LIN {X 0,Y 141.278,Z 230.592,A -85,B 0,C 180,E1 -25855.05,E2 -25855.05} C_VEL
LIN {X 0,Y 135.258,Z 217.256,A -85,B 0,C 180,E1 -25857.958,E2 -25857.958} C_VEL
LIN {X 0,Y 129.274,Z 206.453,A -85,B 0,C 180,E1 -25861.051,E2 -25861.051} C_VEL
LIN {X 0,Y 124.836,Z 199.374,A -85,B 0,C 180,E1 -25863.554,E2 -25863.554} C_VEL
LIN {X 0,Y 120.846,Z 193.414,A -85,B 0,C 180,E1 -25866.03,E2 -25866.03} C_VEL
LIN {X 0,Y 118.527,Z 190.076,A -85,B 0,C 180,E1 -25867.593,E2 -25867.593} C_VEL
LIN {X 0,Y 118.058,Z 189.3,A -85,B 0,C 180,E1 -25867.932,E2 -25867.932} C_VEL
LIN {X 0,Y 115.859,Z 187.104,A -85,B 0,C 180,E1 -25869.449,E2 -25869.449} C_VEL
LIN {X 0,Y 114.927,Z 184.823,A -85,B 0,C 180,E1 -25870.265,E2 -25870.265} C_VEL
LIN {X 0,Y 114.809,Z 184.184,A -85,B 0,C 180,E1 -25870.536,E2 -25870.536} C_VEL
LIN {X 0,Y 114.767,Z 184.142,A -85,B 0,C 180,E1 -25877.657,E2 -25877.657} C_VEL
LIN {X 0,Y 114.783,Z 184.185,A -85,B 0,C 180,E1 -25882.749,E2 -25882.749} C_VEL
LIN {X 0,Y 114.839,Z 184.117,A -85,B 0,C 180,E1 -25888.959,E2 -25888.959} C_VEL
LIN {X 0,Y 114.899,Z 184.166,A -85,B 0,C 180,E1 -25896.566,E2 -25896.566} C_VEL
LIN {X 0,Y 114.963,Z 184.147,A -85,B 0,C 180,E1 -25902.204,E2 -25902.204} C_VEL
LIN {X 0,Y 115.306,Z 184.11,A -85,B 0,C 180,E1 -25909.466,E2 -25909.466} C_VEL
LIN {X 0,Y 115.487,Z 184.099,A -85,B 0,C 180,E1 -25916.513,E2 -25916.513} C_VEL
LIN {X 0,Y 115.951,Z 184.025,A -85,B 0,C 180,E1 -25920.002,E2 -25920.002} C_VEL
LIN {X 0,Y 115.351,Z 184.103,A -85,B 0,C 180,E1 -25927.001,E2 -25927.001} C_VEL
LIN {X 0,Y 115.207,Z 184.136,A -85,B 0,C 180,E1 -25932.559,E2 -25932.559} C_VEL
LIN {X 0,Y 114.969,Z 184.154,A -85,B 0,C 180,E1 -25937.799,E2 -25937.799} C_VEL
LIN {X 0,Y 114.914,Z 184.172,A -85,B 0,C 180,E1 -25943.451,E2 -25943.451} C_VEL
LIN {X 0,Y 114.863,Z 184.178,A -85,B 0,C 180,E1 -25949.058,E2 -25949.058} C_VEL
LIN {X 0,Y 115.85,Z 186.976,A -85,B 0,C 180,E1 -25950.008,E2 -25950.008} C_VEL
LIN {X 0,Y 117.94,Z 189.165,A -85,B 0,C 180,E1 -25951.46,E2 -25951.46} C_VEL
LIN {X 0,Y 118.811,Z 190.602,A -85,B 0,C 180,E1 -25952.087,E2 -25952.087} C_VEL
LIN {X 0,Y 121.086,Z 193.68,A -85,B 0,C 180,E1 -25953.59,E2 -25953.59} C_VEL
LIN {X 0,Y 126.955,Z 202.682,A -85,B 0,C 180,E1 -25957.142,E2 -25957.142} C_VEL
LIN {X 0,Y 130.736,Z 209.225,A -85,B 0,C 180,E1 -25959.227,E2 -25959.227} C_VEL
LIN {X 0,Y 135.81,Z 221.695,A -85,B 0,C 180,E1 -25962.03,E2 -25962.03} C_VEL
LIN {X 0,Y 139.584,Z 233.149,A -85,B 0,C 180,E1 -25964.065,E2 -25964.065} C_VEL
LIN {X 0,Y 140.517,Z 245.678,A -85,B 0,C 180,E1 -25965.174,E2 -25965.174} C_VEL
LIN {X 0,Y 137.592,Z 288.137,A -85,B 0,C 180,E1 -25967.172,E2 -25967.172} C_VEL
LIN {X 0,Y 135.71,Z 301.694,A -85,B 0,C 180,E1 -25968.306,E2 -25968.306} C_VEL
LIN {X 0,Y 133.388,Z 313.543,A -85,B 0,C 180,E1 -25969.801,E2 -25969.801} C_VEL
LIN {X 0,Y 130.614,Z 324.787,A -85,B 0,C 180,E1 -25971.772,E2 -25971.772} C_VEL
LIN {X 0,Y 127.55,Z 335.152,A -85,B 0,C 180,E1 -25974.165,E2 -25974.165} C_VEL
LIN {X 0,Y 124.027,Z 345.896,A -85,B 0,C 180,E1 -25977.43,E2 -25977.43} C_VEL
LIN {X 0,Y 121.167,Z 354.142,A -85,B 0,C 180,E1 -25980.656,E2 -25980.656} C_VEL
LIN {X 0,Y 117.858,Z 363.477,A -85,B 0,C 180,E1 -25985.328,E2 -25985.328} C_VEL
LIN {X 0,Y 115.267,Z 371.169,A -85,B 0,C 180,E1 -25990.406,E2 -25990.406} C_VEL
LIN {X 0,Y 113.501,Z 377.329,A -85,B 0,C 180,E1 -25995.659,E2 -25995.659} C_VEL
LIN {X 0,Y 112.596,Z 382.185,A -85,B 0,C 180,E1 -26001.022,E2 -26001.022} C_VEL
LIN {X 0,Y 112.341,Z 385.87,A -85,B 0,C 180,E1 -26006.413,E2 -26006.413} C_VEL
LIN {X 0,Y 112.454,Z 387.919,A -85,B 0,C 180,E1 -26010.362,E2 -26010.362} C_VEL
LIN {X 0,Y 112.336,Z 389.142,A -85,B 0,C 180,E1 -26013.586,E2 -26013.586} C_VEL
LIN {X 0,Y 112.831,Z 390.682,A -85,B 0,C 180,E1 -26020.769,E2 -26020.769} C_VEL
LIN {X 0,Y 114.797,Z 390.713,A -85,B 0,C 180,E1 -26027.824,E2 -26027.824} C_VEL
LIN {X 0,Y 118.532,Z 389.166,A -85,B 0,C 180,E1 -26034.522,E2 -26034.522} C_VEL
LIN {X 0,Y 123.893,Z 386.089,A -85,B 0,C 180,E1 -26040.699,E2 -26040.699} C_VEL
LIN {X 0,Y 128.757,Z 382.601,A -85,B 0,C 180,E1 -26045.037,E2 -26045.037} C_VEL
LIN {X 0,Y 135.201,Z 377.315,A -85,B 0,C 180,E1 -26049.537,E2 -26049.537} C_VEL
LIN {X 0,Y 141.582,Z 371.476,A -85,B 0,C 180,E1 -26053.042,E2 -26053.042} C_VEL
LIN {X 0,Y 145.984,Z 367,A -85,B 0,C 180,E1 -26055.088,E2 -26055.088} C_VEL
LIN {X 0,Y 148.771,Z 363.579,A -85,B 0,C 180,E1 -26056.614,E2 -26056.614} C_VEL
LIN {X 0,Y 151.909,Z 357.771,A -85,B 0,C 180,E1 -26059.441,E2 -26059.441} C_VEL
LIN {X 0,Y 155.058,Z 351.474,A -85,B 0,C 180,E1 -26062.04,E2 -26062.04} C_VEL
LIN {X 0,Y 157.739,Z 347.223,A -85,B 0,C 180,E1 -26063.181,E2 -26063.181} C_VEL
LIN {X 0,Y 164.092,Z 337.097,A -85,B 0,C 180,E1 -26064.996,E2 -26064.996} C_VEL
LIN {X 0,Y 169.797,Z 326.151,A -85,B 0,C 180,E1 -26066.406,E2 -26066.406} C_VEL
LIN {X 0,Y 174.86,Z 313.961,A -85,B 0,C 180,E1 -26067.569,E2 -26067.569} C_VEL
LIN {X 0,Y 178.951,Z 301.013,A -85,B 0,C 180,E1 -26068.419,E2 -26068.419} C_VEL
LIN {X 0,Y 181.772,Z 287.524,A -85,B 0,C 180,E1 -26069.046,E2 -26069.046} C_VEL
LIN {X 0,Y 183.069,Z 276.561,A -85,B 0,C 180,E1 -26069.451,E2 -26069.451} C_VEL
LIN {X 0,Y 180.59,Z 269.148,A -85,B 0,C 180,E1 -26072.395,E2 -26072.395} C_VEL
LIN {X 0,Y 178.521,Z 263.589,A -85,B 0,C 180,E1 -26075.281,E2 -26075.281} C_VEL
LIN {X 0,Y 177.22,Z 260.269,A -85,B 0,C 180,E1 -26077.406,E2 -26077.406} C_VEL
LIN {X 0,Y 175.668,Z 256.541,A -85,B 0,C 180,E1 -26080.476,E2 -26080.476} C_VEL
LIN {X 0,Y 173.962,Z 252.285,A -85,B 0,C 180,E1 -26086.388,E2 -26086.388} C_VEL
LIN {X 0,Y 173.776,Z 252.037,A -85,B 0,C 180,E1 -26093.03,E2 -26093.03} C_VEL
LIN {X 0,Y 174.336,Z 252.524,A -85,B 0,C 180,E1 -26095.701,E2 -26095.701} C_VEL
LIN {X 0,Y 175.835,Z 256.038,A -85,B 0,C 180,E1 -26100.247,E2 -26100.247} C_VEL
LIN {X 0,Y 176.48,Z 257.185,A -85,B 0,C 180,E1 -26101.532,E2 -26101.532} C_VEL
LIN {X 0,Y 178.026,Z 260.23,A -85,B 0,C 180,E1 -26104.164,E2 -26104.164} C_VEL
LIN {X 0,Y 180.321,Z 264.764,A -85,B 0,C 180,E1 -26107.327,E2 -26107.327} C_VEL
LIN {X 0,Y 183.501,Z 271.507,A -85,B 0,C 180,E1 -26110.899,E2 -26110.899} C_VEL
LIN {X 0,Y 183.126,Z 276.091,A -85,B 0,C 180,E1 -26111.124,E2 -26111.124} C_VEL
LIN {X 0,Y 180.943,Z 289.564,A -85,B 0,C 180,E1 -26111.653,E2 -26111.653} C_VEL
LIN {X 0,Y 177.684,Z 302.377,A -85,B 0,C 180,E1 -26112.452,E2 -26112.452} C_VEL
LIN {X 0,Y 173.505,Z 314.371,A -85,B 0,C 180,E1 -26113.555,E2 -26113.555} C_VEL
LIN {X 0,Y 168.375,Z 325.796,A -85,B 0,C 180,E1 -26114.944,E2 -26114.944} C_VEL
LIN {X 0,Y 162.34,Z 336.631,A -85,B 0,C 180,E1 -26116.698,E2 -26116.698} C_VEL
LIN {X 0,Y 155.887,Z 346.195,A -85,B 0,C 180,E1 -26118.78,E2 -26118.78} C_VEL
LIN {X 0,Y 148.997,Z 354.873,A -85,B 0,C 180,E1 -26121.319,E2 -26121.319} C_VEL
LIN {X 0,Y 142.4,Z 361.96,A -85,B 0,C 180,E1 -26124.071,E2 -26124.071} C_VEL
LIN {X 0,Y 134.979,Z 368.819,A -85,B 0,C 180,E1 -26127.731,E2 -26127.731} C_VEL
LIN {X 0,Y 128.163,Z 374.126,A -85,B 0,C 180,E1 -26131.793,E2 -26131.793} C_VEL
LIN {X 0,Y 122.071,Z 378.141,A -85,B 0,C 180,E1 -26136.291,E2 -26136.291} C_VEL
LIN {X 0,Y 116.436,Z 381.145,A -85,B 0,C 180,E1 -26141.599,E2 -26141.599} C_VEL
LIN {X 0,Y 112.44,Z 382.723,A -85,B 0,C 180,E1 -26146.564,E2 -26146.564} C_VEL
LIN {X 0,Y 110.07,Z 383.318,A -85,B 0,C 180,E1 -26150.32,E2 -26150.32} C_VEL
LIN {X 0,Y 108.113,Z 383.454,A -85,B 0,C 180,E1 -26154.194,E2 -26154.194} C_VEL
LIN {X 0,Y 106.34,Z 382.966,A -85,B 0,C 180,E1 -26159.219,E2 -26159.219} C_VEL
LIN {X 0,Y 104.953,Z 381.137,A -85,B 0,C 180,E1 -26166.311,E2 -26166.311} C_VEL
LIN {X 0,Y 104.829,Z 378.437,A -85,B 0,C 180,E1 -26172.441,E2 -26172.441} C_VEL
LIN {X 0,Y 105.527,Z 374.657,A -85,B 0,C 180,E1 -26178.475,E2 -26178.475} C_VEL
LIN {X 0,Y 106.954,Z 369.712,A -85,B 0,C 180,E1 -26184.344,E2 -26184.344} C_VEL
LIN {X 0,Y 109.063,Z 363.479,A -85,B 0,C 180,E1 -26190.001,E2 -26190.001} C_VEL
LIN {X 0,Y 112.006,Z 355.718,A -85,B 0,C 180,E1 -26195.401,E2 -26195.401} C_VEL
LIN {X 0,Y 115.134,Z 347.56,A -85,B 0,C 180,E1 -26199.773,E2 -26199.773} C_VEL
LIN {X 0,Y 119.047,Z 336.935,A -85,B 0,C 180,E1 -26204.095,E2 -26204.095} C_VEL
LIN {X 0,Y 122.703,Z 325.882,A -85,B 0,C 180,E1 -26207.501,E2 -26207.501} C_VEL
LIN {X 0,Y 125.845,Z 315.014,A -85,B 0,C 180,E1 -26210.003,E2 -26210.003} C_VEL
LIN {X 0,Y 128.563,Z 303.148,A -85,B 0,C 180,E1 -26212.076,E2 -26212.076} C_VEL
LIN {X 0,Y 130.799,Z 290.5,A -85,B 0,C 180,E1 -26213.651,E2 -26213.651} C_VEL
LIN {X 0,Y 132.401,Z 277.456,A -85,B 0,C 180,E1 -26214.67,E2 -26214.67} C_VEL
LIN {X 0,Y 135.487,Z 232.577,A -85,B 0,C 180,E1 -26216.802,E2 -26216.802} C_VEL
LIN {X 0,Y 130.033,Z 220.377,A -85,B 0,C 180,E1 -26219.693,E2 -26219.693} C_VEL
LIN {X 0,Y 124.019,Z 209.324,A -85,B 0,C 180,E1 -26223.102,E2 -26223.102} C_VEL
LIN {X 0,Y 119.218,Z 201.809,A -85,B 0,C 180,E1 -26226.123,E2 -26226.123} C_VEL
LIN {X 0,Y 116.893,Z 198.387,A -85,B 0,C 180,E1 -26227.725,E2 -26227.725} C_VEL
LIN {X 0,Y 114.59,Z 194.971,A -85,B 0,C 180,E1 -26229.434,E2 -26229.434} C_VEL
LIN {X 0,Y 112.355,Z 192.252,A -85,B 0,C 180,E1 -26231.161,E2 -26231.161} C_VEL
LIN {X 0,Y 111.209,Z 190.299,A -85,B 0,C 180,E1 -26232.152,E2 -26232.152} C_VEL
LIN {X 0,Y 108.801,Z 188.128,A -85,B 0,C 180,E1 -26234.158,E2 -26234.158} C_VEL
LIN {X 0,Y 107.714,Z 185.508,A -85,B 0,C 180,E1 -26235.33,E2 -26235.33} C_VEL
LIN {X 0,Y 107.641,Z 185.029,A -85,B 0,C 180,E1 -26235.553,E2 -26235.553} C_VEL
LIN {X 0,Y 107.68,Z 185.063,A -85,B 0,C 180,E1 -26241.557,E2 -26241.557} C_VEL
LIN {X 0,Y 107.777,Z 184.997,A -85,B 0,C 180,E1 -26248.558,E2 -26248.558} C_VEL
LIN {X 0,Y 107.866,Z 185.044,A -85,B 0,C 180,E1 -26256.99,E2 -26256.99} C_VEL
LIN {X 0,Y 107.86,Z 185.036,A -85,B 0,C 180,E1 -26260.989,E2 -26260.989} C_VEL
LIN {X 0,Y 108.206,Z 184.999,A -85,B 0,C 180,E1 -26268.766,E2 -26268.766} C_VEL
LIN {X 0,Y 108.288,Z 184.982,A -85,B 0,C 180,E1 -26272.544,E2 -26272.544} C_VEL
LIN {X 0,Y 108.88,Z 184.906,A -85,B 0,C 180,E1 -26280.002,E2 -26280.002} C_VEL
LIN {X 0,Y 108.29,Z 184.98,A -85,B 0,C 180,E1 -26287.46,E2 -26287.46} C_VEL
LIN {X 0,Y 108.141,Z 185.015,A -85,B 0,C 180,E1 -26292.874,E2 -26292.874} C_VEL
LIN {X 0,Y 107.866,Z 185.048,A -85,B 0,C 180,E1 -26299.015,E2 -26299.015} C_VEL
LIN {X 0,Y 107.843,Z 185.082,A -85,B 0,C 180,E1 -26304.209,E2 -26304.209} C_VEL
LIN {X 0,Y 108.633,Z 187.607,A -85,B 0,C 180,E1 -26305.138,E2 -26305.138} C_VEL
LIN {X 0,Y 110.661,Z 189.893,A -85,B 0,C 180,E1 -26306.906,E2 -26306.906} C_VEL
LIN {X 0,Y 111.629,Z 190.672,A -85,B 0,C 180,E1 -26307.668,E2 -26307.668} C_VEL
LIN {X 0,Y 113.696,Z 194.04,A -85,B 0,C 180,E1 -26309.385,E2 -26309.385} C_VEL
LIN {X 0,Y 115.23,Z 195.866,A -85,B 0,C 180,E1 -26310.523,E2 -26310.523} C_VEL
LIN {X 0,Y 118.775,Z 201.22,A -85,B 0,C 180,E1 -26313.06,E2 -26313.06} C_VEL
LIN {X 0,Y 122.699,Z 207.23,A -85,B 0,C 180,E1 -26315.576,E2 -26315.576} C_VEL
LIN {X 0,Y 126.312,Z 213.657,A -85,B 0,C 180,E1 -26317.739,E2 -26317.739} C_VEL
LIN {X 0,Y 131.202,Z 226.135,A -85,B 0,C 180,E1 -26320.671,E2 -26320.671} C_VEL
LIN {X 0,Y 134.166,Z 235.753,A -85,B 0,C 180,E1 -26322.444,E2 -26322.444} C_VEL
LIN {X 0,Y 134.842,Z 246.309,A -85,B 0,C 180,E1 -26323.411,E2 -26323.411} C_VEL
LIN {X 0,Y 131.886,Z 287.406,A -85,B 0,C 180,E1 -26325.382,E2 -26325.382} C_VEL
LIN {X 0,Y 129.94,Z 301.041,A -85,B 0,C 180,E1 -26326.534,E2 -26326.534} C_VEL
LIN {X 0,Y 127.521,Z 312.999,A -85,B 0,C 180,E1 -26328.067,E2 -26328.067} C_VEL
LIN {X 0,Y 124.61,Z 324.325,A -85,B 0,C 180,E1 -26330.092,E2 -26330.092} C_VEL
LIN {X 0,Y 121.37,Z 334.721,A -85,B 0,C 180,E1 -26332.553,E2 -26332.553} C_VEL
LIN {X 0,Y 118.021,Z 344.404,A -85,B 0,C 180,E1 -26335.547,E2 -26335.547} C_VEL
LIN {X 0,Y 115.432,Z 351.869,A -85,B 0,C 180,E1 -26338.475,E2 -26338.475} C_VEL
LIN {X 0,Y 113.081,Z 357.698,A -85,B 0,C 180,E1 -26341.205,E2 -26341.205} C_VEL
LIN {X 0,Y 109.924,Z 366.571,A -85,B 0,C 180,E1 -26346.446,E2 -26346.446} C_VEL
LIN {X 0,Y 107.418,Z 373.582,A -85,B 0,C 180,E1 -26351.893,E2 -26351.893} C_VEL
LIN {X 0,Y 105.812,Z 380.007,A -85,B 0,C 180,E1 -26358.506,E2 -26358.506} C_VEL
LIN {X 0,Y 105.278,Z 384.176,A -85,B 0,C 180,E1 -26364.252,E2 -26364.252} C_VEL
LIN {X 0,Y 105.408,Z 387.241,A -85,B 0,C 180,E1 -26369.999,E2 -26369.999} C_VEL
LIN {X 0,Y 105.246,Z 388.707,A -85,B 0,C 180,E1 -26373.828,E2 -26373.828} C_VEL
LIN {X 0,Y 105.343,Z 389.727,A -85,B 0,C 180,E1 -26377.667,E2 -26377.667} C_VEL
LIN {X 0,Y 106.726,Z 390.602,A -85,B 0,C 180,E1 -26385.272,E2 -26385.272} C_VEL
LIN {X 0,Y 109.802,Z 389.978,A -85,B 0,C 180,E1 -26392.583,E2 -26392.583} C_VEL
LIN {X 0,Y 114.756,Z 387.774,A -85,B 0,C 180,E1 -26399.336,E2 -26399.336} C_VEL
LIN {X 0,Y 119.486,Z 385.087,A -85,B 0,C 180,E1 -26403.971,E2 -26403.971} C_VEL
LIN {X 0,Y 124.793,Z 381.433,A -85,B 0,C 180,E1 -26408.278,E2 -26408.278} C_VEL
LIN {X 0,Y 130.885,Z 376.711,A -85,B 0,C 180,E1 -26412.159,E2 -26412.159} C_VEL
LIN {X 0,Y 138.844,Z 369.661,A -85,B 0,C 180,E1 -26416.162,E2 -26416.162} C_VEL
LIN {X 0,Y 146.16,Z 362.066,A -85,B 0,C 180,E1 -26419.229,E2 -26419.229} C_VEL
LIN {X 0,Y 153.86,Z 352.578,A -85,B 0,C 180,E1 -26421.994,E2 -26421.994} C_VEL
LIN {X 0,Y 157.739,Z 347.223,A -85,B 0,C 180,E1 -26423.181,E2 -26423.181} C_VEL
LIN {X 0,Y 160.416,Z 342.829,A -85,B 0,C 180,E1 -26424.228,E2 -26424.228} C_VEL
LIN {X 0,Y 163.562,Z 335.484,A -85,B 0,C 180,E1 -26426.305,E2 -26426.305} C_VEL
LIN {X 0,Y 166.376,Z 327.705,A -85,B 0,C 180,E1 -26428.198,E2 -26428.198} C_VEL
LIN {X 0,Y 168.442,Z 322.634,A -85,B 0,C 180,E1 -26428.95,E2 -26428.95} C_VEL
LIN {X 0,Y 173.404,Z 310.062,A -85,B 0,C 180,E1 -26429.999,E2 -26429.999} C_VEL
LIN {X 0,Y 177.23,Z 297.039,A -85,B 0,C 180,E1 -26430.739,E2 -26430.739} C_VEL
LIN {X 0,Y 179.618,Z 284.687,A -85,B 0,C 180,E1 -26431.246,E2 -26431.246} C_VEL
LIN {X 0,Y 180.154,Z 279.887,A -85,B 0,C 180,E1 -26431.456,E2 -26431.456} C_VEL
LIN {X 0,Y 177.91,Z 272.769,A -85,B 0,C 180,E1 -26434.603,E2 -26434.603} C_VEL
LIN {X 0,Y 176.019,Z 267.262,A -85,B 0,C 180,E1 -26437.785,E2 -26437.785} C_VEL
LIN {X 0,Y 174.427,Z 263.199,A -85,B 0,C 180,E1 -26441.194,E2 -26441.194} C_VEL
LIN {X 0,Y 172.994,Z 259.277,A -85,B 0,C 180,E1 -26446.729,E2 -26446.729} C_VEL
LIN {X 0,Y 172.871,Z 259.051,A -85,B 0,C 180,E1 -26452.993,E2 -26452.993} C_VEL
LIN {X 0,Y 173.33,Z 259.539,A -85,B 0,C 180,E1 -26455.347,E2 -26455.347} C_VEL
LIN {X 0,Y 174.662,Z 262.838,A -85,B 0,C 180,E1 -26459.711,E2 -26459.711} C_VEL
LIN {X 0,Y 175.334,Z 264.232,A -85,B 0,C 180,E1 -26461.187,E2 -26461.187} C_VEL
LIN {X 0,Y 176.665,Z 267.032,A -85,B 0,C 180,E1 -26463.586,E2 -26463.586} C_VEL
LIN {X 0,Y 178.604,Z 271.098,A -85,B 0,C 180,E1 -26466.447,E2 -26466.447} C_VEL
LIN {X 0,Y 180.587,Z 275.57,A -85,B 0,C 180,E1 -26468.954,E2 -26468.954} C_VEL
LIN {X 0,Y 179.677,Z 282.6,A -85,B 0,C 180,E1 -26469.248,E2 -26469.248} C_VEL
LIN {X 0,Y 176.935,Z 295.608,A -85,B 0,C 180,E1 -26469.855,E2 -26469.855} C_VEL
LIN {X 0,Y 173.041,Z 308.336,A -85,B 0,C 180,E1 -26470.779,E2 -26470.779} C_VEL
LIN {X 0,Y 167.948,Z 320.78,A -85,B 0,C 180,E1 -26472.076,E2 -26472.076} C_VEL
LIN {X 0,Y 162.595,Z 331.095,A -85,B 0,C 180,E1 -26473.458,E2 -26473.458} C_VEL
LIN {X 0,Y 156.593,Z 340.738,A -85,B 0,C 180,E1 -26475.188,E2 -26475.188} C_VEL
LIN {X 0,Y 149.238,Z 350.492,A -85,B 0,C 180,E1 -26477.518,E2 -26477.518} C_VEL
LIN {X 0,Y 141.568,Z 359.059,A -85,B 0,C 180,E1 -26480.333,E2 -26480.333} C_VEL
LIN {X 0,Y 134.144,Z 366.093,A -85,B 0,C 180,E1 -26483.531,E2 -26483.531} C_VEL
LIN {X 0,Y 126.617,Z 372.071,A -85,B 0,C 180,E1 -26487.365,E2 -26487.365} C_VEL
LIN {X 0,Y 119.375,Z 376.925,A -85,B 0,C 180,E1 -26491.994,E2 -26491.994} C_VEL
LIN {X 0,Y 113.684,Z 380.057,A -85,B 0,C 180,E1 -26496.519,E2 -26496.519} C_VEL
LIN {X 0,Y 110.102,Z 381.693,A -85,B 0,C 180,E1 -26500.006,E2 -26500.006} C_VEL
LIN {X 0,Y 106.977,Z 382.829,A -85,B 0,C 180,E1 -26503.726,E2 -26503.726} C_VEL
LIN {X 0,Y 103.954,Z 383.544,A -85,B 0,C 180,E1 -26508.042,E2 -26508.042} C_VEL
LIN {X 0,Y 101.973,Z 383.73,A -85,B 0,C 180,E1 -26511.664,E2 -26511.664} C_VEL
LIN {X 0,Y 99.547,Z 383.226,A -85,B 0,C 180,E1 -26517.904,E2 -26517.904} C_VEL
LIN {X 0,Y 98.055,Z 381.687,A -85,B 0,C 180,E1 -26524.53,E2 -26524.53} C_VEL
LIN {X 0,Y 97.695,Z 379.954,A -85,B 0,C 180,E1 -26529.254,E2 -26529.254} C_VEL
LIN {X 0,Y 97.965,Z 376.841,A -85,B 0,C 180,E1 -26535.459,E2 -26535.459} C_VEL
LIN {X 0,Y 99.252,Z 371.984,A -85,B 0,C 180,E1 -26542.433,E2 -26542.433} C_VEL
LIN {X 0,Y 101.349,Z 365.814,A -85,B 0,C 180,E1 -26549.007,E2 -26549.007} C_VEL
LIN {X 0,Y 104.205,Z 358.544,A -85,B 0,C 180,E1 -26554.837,E2 -26554.837} C_VEL
LIN {X 0,Y 107.597,Z 350.189,A -85,B 0,C 180,E1 -26559.925,E2 -26559.925} C_VEL
LIN {X 0,Y 111.205,Z 341.099,A -85,B 0,C 180,E1 -26564.176,E2 -26564.176} C_VEL
LIN {X 0,Y 114.978,Z 330.966,A -85,B 0,C 180,E1 -26567.797,E2 -26567.797} C_VEL
LIN {X 0,Y 118.569,Z 319.706,A -85,B 0,C 180,E1 -26570.834,E2 -26570.834} C_VEL
LIN {X 0,Y 121.889,Z 307.108,A -85,B 0,C 180,E1 -26573.355,E2 -26573.355} C_VEL
LIN {X 0,Y 124.369,Z 295.557,A -85,B 0,C 180,E1 -26574.987,E2 -26574.987} C_VEL
LIN {X 0,Y 126.211,Z 282.571,A -85,B 0,C 180,E1 -26576.269,E2 -26576.269} C_VEL
LIN {X 0,Y 127.78,Z 264.618,A -85,B 0,C 180,E1 -26577.243,E2 -26577.243} C_VEL
LIN {X 0,Y 129.923,Z 234.688,A -85,B 0,C 180,E1 -26578.664,E2 -26578.664} C_VEL
LIN {X 0,Y 125.292,Z 224.298,A -85,B 0,C 180,E1 -26581.317,E2 -26581.317} C_VEL
LIN {X 0,Y 119.759,Z 213.837,A -85,B 0,C 180,E1 -26584.759,E2 -26584.759} C_VEL
LIN {X 0,Y 114.032,Z 204.534,A -85,B 0,C 180,E1 -26588.807,E2 -26588.807} C_VEL
LIN {X 0,Y 110.929,Z 200.241,A -85,B 0,C 180,E1 -26591.259,E2 -26591.259} C_VEL
LIN {X 0,Y 108.21,Z 196.314,A -85,B 0,C 180,E1 -26593.643,E2 -26593.643} C_VEL
LIN {X 0,Y 105.695,Z 193.536,A -85,B 0,C 180,E1 -26595.984,E2 -26595.984} C_VEL
LIN {X 0,Y 104.735,Z 191.517,A -85,B 0,C 180,E1 -26597.073,E2 -26597.073} C_VEL
LIN {X 0,Y 102.17,Z 189.554,A -85,B 0,C 180,E1 -26599.762,E2 -26599.762} C_VEL
LIN {X 0,Y 100.96,Z 187.325,A -85,B 0,C 180,E1 -26601.37,E2 -26601.37} C_VEL
LIN {X 0,Y 100.637,Z 185.943,A -85,B 0,C 180,E1 -26602.02,E2 -26602.02} C_VEL
LIN {X 0,Y 100.68,Z 185.895,A -85,B 0,C 180,E1 -26606.896,E2 -26606.896} C_VEL
LIN {X 0,Y 100.724,Z 185.91,A -85,B 0,C 180,E1 -26615.253,E2 -26615.253} C_VEL
LIN {X 0,Y 100.775,Z 185.928,A -85,B 0,C 180,E1 -26619.595,E2 -26619.595} C_VEL
LIN {X 0,Y 101.116,Z 185.888,A -85,B 0,C 180,E1 -26627.967,E2 -26627.967} C_VEL
LIN {X 0,Y 101.222,Z 185.859,A -85,B 0,C 180,E1 -26632.02,E2 -26632.02} C_VEL
LIN {X 0,Y 101.812,Z 185.785,A -85,B 0,C 180,E1 -26640.002,E2 -26640.002} C_VEL
LIN {X 0,Y 101.227,Z 185.859,A -85,B 0,C 180,E1 -26647.984,E2 -26647.984} C_VEL
LIN {X 0,Y 101.053,Z 185.896,A -85,B 0,C 180,E1 -26653.174,E2 -26653.174} C_VEL
LIN {X 0,Y 100.822,Z 186.076,A -85,B 0,C 180,E1 -26657.759,E2 -26657.759} C_VEL
LIN {X 0,Y 101.579,Z 188.351,A -85,B 0,C 180,E1 -26658.926,E2 -26658.926} C_VEL
LIN {X 0,Y 103.281,Z 190.508,A -85,B 0,C 180,E1 -26660.933,E2 -26660.933} C_VEL
LIN {X 0,Y 104.982,Z 191.722,A -85,B 0,C 180,E1 -26662.642,E2 -26662.642} C_VEL
LIN {X 0,Y 106.67,Z 194.691,A -85,B 0,C 180,E1 -26664.442,E2 -26664.442} C_VEL
LIN {X 0,Y 108.801,Z 197.031,A -85,B 0,C 180,E1 -26666.367,E2 -26666.367} C_VEL
LIN {X 0,Y 111.465,Z 200.746,A -85,B 0,C 180,E1 -26668.641,E2 -26668.641} C_VEL
LIN {X 0,Y 116.879,Z 209.108,A -85,B 0,C 180,E1 -26672.766,E2 -26672.766} C_VEL
LIN {X 0,Y 121.736,Z 217.59,A -85,B 0,C 180,E1 -26676.005,E2 -26676.005} C_VEL
LIN {X 0,Y 126.3,Z 229.61,A -85,B 0,C 180,E1 -26678.996,E2 -26678.996} C_VEL
LIN {X 0,Y 128.805,Z 238.06,A -85,B 0,C 180,E1 -26680.642,E2 -26680.642} C_VEL
LIN {X 0,Y 129.276,Z 247.345,A -85,B 0,C 180,E1 -26681.515,E2 -26681.515} C_VEL
LIN {X 0,Y 126.167,Z 287.86,A -85,B 0,C 180,E1 -26683.513,E2 -26683.513} C_VEL
LIN {X 0,Y 124.161,Z 301.141,A -85,B 0,C 180,E1 -26684.675,E2 -26684.675} C_VEL
LIN {X 0,Y 121.501,Z 313.543,A -85,B 0,C 180,E1 -26686.329,E2 -26686.329} C_VEL
LIN {X 0,Y 118.213,Z 325.453,A -85,B 0,C 180,E1 -26688.592,E2 -26688.592} C_VEL
LIN {X 0,Y 114.897,Z 335.615,A -85,B 0,C 180,E1 -26691.172,E2 -26691.172} C_VEL
LIN {X 0,Y 111.388,Z 345.097,A -85,B 0,C 180,E1 -26694.293,E2 -26694.293} C_VEL
LIN {X 0,Y 108.01,Z 353.727,A -85,B 0,C 180,E1 -26697.968,E2 -26697.968} C_VEL
LIN {X 0,Y 104.426,Z 362.775,A -85,B 0,C 180,E1 -26702.98,E2 -26702.98} C_VEL
LIN {X 0,Y 101.483,Z 370.506,A -85,B 0,C 180,E1 -26708.679,E2 -26708.679} C_VEL
LIN {X 0,Y 99.206,Z 377.608,A -85,B 0,C 180,E1 -26715.643,E2 -26715.643} C_VEL
LIN {X 0,Y 98.331,Z 382.289,A -85,B 0,C 180,E1 -26721.781,E2 -26721.781} C_VEL
LIN {X 0,Y 98.173,Z 384.747,A -85,B 0,C 180,E1 -26725.894,E2 -26725.894} C_VEL
LIN {X 0,Y 98.315,Z 386.728,A -85,B 0,C 180,E1 -26729.999,E2 -26729.999} C_VEL
LIN {X 0,Y 98.186,Z 388.244,A -85,B 0,C 180,E1 -26734.104,E2 -26734.104} C_VEL
LIN {X 0,Y 98.296,Z 389.346,A -85,B 0,C 180,E1 -26738.221,E2 -26738.221} C_VEL
LIN {X 0,Y 99.855,Z 390.316,A -85,B 0,C 180,E1 -26746.351,E2 -26746.351} C_VEL
LIN {X 0,Y 103.271,Z 389.801,A -85,B 0,C 180,E1 -26754.099,E2 -26754.099} C_VEL
LIN {X 0,Y 105.757,Z 388.975,A -85,B 0,C 180,E1 -26757.721,E2 -26757.721} C_VEL
LIN {X 0,Y 111.916,Z 386.103,A -85,B 0,C 180,E1 -26764.414,E2 -26764.414} C_VEL
LIN {X 0,Y 116.48,Z 383.427,A -85,B 0,C 180,E1 -26768.334,E2 -26768.334} C_VEL
LIN {X 0,Y 123.492,Z 378.633,A -85,B 0,C 180,E1 -26773.072,E2 -26773.072} C_VEL
LIN {X 0,Y 131.586,Z 372.24,A -85,B 0,C 180,E1 -26777.255,E2 -26777.255} C_VEL
LIN {X 0,Y 139.102,Z 365.308,A -85,B 0,C 180,E1 -26780.398,E2 -26780.398} C_VEL
LIN {X 0,Y 145.64,Z 358.271,A -85,B 0,C 180,E1 -26782.771,E2 -26782.771} C_VEL
LIN {X 0,Y 152.387,Z 349.82,A -85,B 0,C 180,E1 -26784.947,E2 -26784.947} C_VEL
LIN {X 0,Y 159.441,Z 339.416,A -85,B 0,C 180,E1 -26786.877,E2 -26786.877} C_VEL
LIN {X 0,Y 166.011,Z 327.731,A -85,B 0,C 180,E1 -26788.428,E2 -26788.428} C_VEL
LIN {X 0,Y 168.442,Z 322.634,A -85,B 0,C 180,E1 -26788.95,E2 -26788.95} C_VEL
LIN {X 0,Y 170.418,Z 317.439,A -85,B 0,C 180,E1 -26789.634,E2 -26789.634} C_VEL
LIN {X 0,Y 172.654,Z 308.903,A -85,B 0,C 180,E1 -26791.14,E2 -26791.14} C_VEL
LIN {X 0,Y 174.362,Z 300.106,A -85,B 0,C 180,E1 -26792.529,E2 -26792.529} C_VEL
LIN {X 0,Y 175.445,Z 294.505,A -85,B 0,C 180,E1 -26793.031,E2 -26793.031} C_VEL
LIN {X 0,Y 177.443,Z 283.563,A -85,B 0,C 180,E1 -26793.467,E2 -26793.467} C_VEL
LIN {X 0,Y 175.874,Z 277.848,A -85,B 0,C 180,E1 -26796.168,E2 -26796.168} C_VEL
LIN {X 0,Y 174.305,Z 273.071,A -85,B 0,C 180,E1 -26799.176,E2 -26799.176} C_VEL
LIN {X 0,Y 173.165,Z 269.703,A -85,B 0,C 180,E1 -26802.077,E2 -26802.077} C_VEL
LIN {X 0,Y 172.004,Z 266.244,A -85,B 0,C 180,E1 -26807.245,E2 -26807.245} C_VEL
LIN {X 0,Y 172.1,Z 266.224,A -85,B 0,C 180,E1 -26813.813,E2 -26813.813} C_VEL
LIN {X 0,Y 172.353,Z 266.683,A -85,B 0,C 180,E1 -26815.134,E2 -26815.134} C_VEL
LIN {X 0,Y 173.899,Z 270.491,A -85,B 0,C 180,E1 -26820.143,E2 -26820.143} C_VEL
LIN {X 0,Y 175.23,Z 273.601,A -85,B 0,C 180,E1 -26822.831,E2 -26822.831} C_VEL
LIN {X 0,Y 177.184,Z 278.093,A -85,B 0,C 180,E1 -26825.999,E2 -26825.999} C_VEL
LIN {X 0,Y 177.825,Z 279.855,A -85,B 0,C 180,E1 -26826.968,E2 -26826.968} C_VEL
LIN {X 0,Y 175.363,Z 292.66,A -85,B 0,C 180,E1 -26827.5,E2 -26827.5} C_VEL
LIN {X 0,Y 171.741,Z 305.187,A -85,B 0,C 180,E1 -26828.293,E2 -26828.293} C_VEL
LIN {X 0,Y 167.52,Z 316.196,A -85,B 0,C 180,E1 -26829.276,E2 -26829.276} C_VEL
LIN {X 0,Y 161.789,Z 327.877,A -85,B 0,C 180,E1 -26830.638,E2 -26830.638} C_VEL
LIN {X 0,Y 155.516,Z 338.116,A -85,B 0,C 180,E1 -26832.24,E2 -26832.24} C_VEL
LIN {X 0,Y 148.625,Z 347.5,A -85,B 0,C 180,E1 -26834.215,E2 -26834.215} C_VEL
LIN {X 0,Y 141.208,Z 356.027,A -85,B 0,C 180,E1 -26836.649,E2 -26836.649} C_VEL
LIN {X 0,Y 132.649,Z 364.224,A -85,B 0,C 180,E1 -26839.876,E2 -26839.876} C_VEL
LIN {X 0,Y 125.556,Z 369.963,A -85,B 0,C 180,E1 -26843.066,E2 -26843.066} C_VEL
LIN {X 0,Y 118.299,Z 374.947,A -85,B 0,C 180,E1 -26846.985,E2 -26846.985} C_VEL
LIN {X 0,Y 111.388,Z 378.887,A -85,B 0,C 180,E1 -26851.595,E2 -26851.595} C_VEL
LIN {X 0,Y 105.088,Z 381.744,A -85,B 0,C 180,E1 -26857.003,E2 -26857.003} C_VEL
LIN {X 0,Y 101.767,Z 382.915,A -85,B 0,C 180,E1 -26860.567,E2 -26860.567} C_VEL
LIN {X 0,Y 97.742,Z 383.822,A -85,B 0,C 180,E1 -26865.971,E2 -26865.971} C_VEL
LIN {X 0,Y 93.926,Z 383.855,A -85,B 0,C 180,E1 -26873.231,E2 -26873.231} C_VEL
LIN {X 0,Y 92.371,Z 383.25,A -85,B 0,C 180,E1 -26877.82,E2 -26877.82} C_VEL
LIN {X 0,Y 91.241,Z 382.205,A -85,B 0,C 180,E1 -26882.474,E2 -26882.474} C_VEL
LIN {X 0,Y 90.609,Z 380.206,A -85,B 0,C 180,E1 -26888.548,E2 -26888.548} C_VEL
LIN {X 0,Y 90.997,Z 376.313,A -85,B 0,C 180,E1 -26896.604,E2 -26896.604} C_VEL
LIN {X 0,Y 92.528,Z 371.188,A -85,B 0,C 180,E1 -26904.124,E2 -26904.124} C_VEL
LIN {X 0,Y 94.969,Z 364.729,A -85,B 0,C 180,E1 -26911.061,E2 -26911.061} C_VEL
LIN {X 0,Y 98.134,Z 357.132,A -85,B 0,C 180,E1 -26917.201,E2 -26917.201} C_VEL
LIN {X 0,Y 101.526,Z 349.367,A -85,B 0,C 180,E1 -26921.987,E2 -26921.987} C_VEL
LIN {X 0,Y 105.485,Z 339.943,A -85,B 0,C 180,E1 -26926.45,E2 -26926.45} C_VEL
LIN {X 0,Y 109.471,Z 329.417,A -85,B 0,C 180,E1 -26930.187,E2 -26930.187} C_VEL
LIN {X 0,Y 113.367,Z 317.711,A -85,B 0,C 180,E1 -26933.28,E2 -26933.28} C_VEL
LIN {X 0,Y 116.456,Z 306.142,A -85,B 0,C 180,E1 -26935.563,E2 -26935.563} C_VEL
LIN {X 0,Y 119.247,Z 292.768,A -85,B 0,C 180,E1 -26937.381,E2 -26937.381} C_VEL
LIN {X 0,Y 121.098,Z 279.552,A -85,B 0,C 180,E1 -26938.565,E2 -26938.565} C_VEL
LIN {X 0,Y 124.437,Z 236.87,A -85,B 0,C 180,E1 -26940.676,E2 -26940.676} C_VEL
LIN {X 0,Y 120.684,Z 228.232,A -85,B 0,C 180,E1 -26943.055,E2 -26943.055} C_VEL
LIN {X 0,Y 115.453,Z 218.048,A -85,B 0,C 180,E1 -26946.652,E2 -26946.652} C_VEL
LIN {X 0,Y 110.309,Z 209.539,A -85,B 0,C 180,E1 -26950.666,E2 -26950.666} C_VEL
LIN {X 0,Y 107.804,Z 205.889,A -85,B 0,C 180,E1 -26952.831,E2 -26952.831} C_VEL
LIN {X 0,Y 105.297,Z 202.257,A -85,B 0,C 180,E1 -26955.206,E2 -26955.206} C_VEL
LIN {X 0,Y 102.627,Z 198.815,A -85,B 0,C 180,E1 -26957.99,E2 -26957.99} C_VEL
LIN {X 0,Y 101.894,Z 197.679,A -85,B 0,C 180,E1 -26958.85,E2 -26958.85} C_VEL
LIN {X 0,Y 99.354,Z 194.995,A -85,B 0,C 180,E1 -26961.925,E2 -26961.925} C_VEL
LIN {X 0,Y 98.13,Z 192.584,A -85,B 0,C 180,E1 -26963.785,E2 -26963.785} C_VEL
LIN {X 0,Y 95.175,Z 190.464,A -85,B 0,C 180,E1 -26968.335,E2 -26968.335} C_VEL
LIN {X 0,Y 93.787,Z 187.888,A -85,B 0,C 180,E1 -26971.314,E2 -26971.314} C_VEL
LIN {X 0,Y 93.56,Z 186.761,A -85,B 0,C 180,E1 -26972.154,E2 -26972.154} C_VEL
LIN {X 0,Y 93.645,Z 186.82,A -85,B 0,C 180,E1 -26977.963,E2 -26977.963} C_VEL
LIN {X 0,Y 94.016,Z 186.775,A -85,B 0,C 180,E1 -26987.043,E2 -26987.043} C_VEL
LIN {X 0,Y 94.133,Z 186.74,A -85,B 0,C 180,E1 -26991.415,E2 -26991.415} C_VEL
LIN {X 0,Y 94.744,Z 186.665,A -85,B 0,C 180,E1 -27000.002,E2 -27000.002} C_VEL
LIN {X 0,Y 94.161,Z 186.896,A -85,B 0,C 180,E1 -27008.587,E2 -27008.587} C_VEL
LIN {X 0,Y 94.819,Z 189.171,A -85,B 0,C 180,E1 -27010.276,E2 -27010.276} C_VEL
LIN {X 0,Y 97.21,Z 191.944,A -85,B 0,C 180,E1 -27014.392,E2 -27014.392} C_VEL
LIN {X 0,Y 98.499,Z 192.812,A -85,B 0,C 180,E1 -27016.186,E2 -27016.186} C_VEL
LIN {X 0,Y 100.218,Z 195.988,A -85,B 0,C 180,E1 -27018.662,E2 -27018.662} C_VEL
LIN {X 0,Y 102.448,Z 198.155,A -85,B 0,C 180,E1 -27021.222,E2 -27021.222} C_VEL
LIN {X 0,Y 104.76,Z 201.613,A -85,B 0,C 180,E1 -27023.738,E2 -27023.738} C_VEL
LIN {X 0,Y 106.084,Z 203.214,A -85,B 0,C 180,E1 -27025.017,E2 -27025.017} C_VEL
LIN {X 0,Y 110.899,Z 210.377,A -85,B 0,C 180,E1 -27029.297,E2 -27029.297} C_VEL
LIN {X 0,Y 116.448,Z 219.933,A -85,B 0,C 180,E1 -27033.548,E2 -27033.548} C_VEL
LIN {X 0,Y 118.638,Z 225.08,A -85,B 0,C 180,E1 -27035.153,E2 -27035.153} C_VEL
LIN {X 0,Y 122.151,Z 235.325,A -85,B 0,C 180,E1 -27037.685,E2 -27037.685} C_VEL
LIN {X 0,Y 123.484,Z 239.843,A -85,B 0,C 180,E1 -27038.632,E2 -27038.632} C_VEL
LIN {X 0,Y 123.812,Z 248.939,A -85,B 0,C 180,E1 -27039.495,E2 -27039.495} C_VEL
LIN {X 0,Y 120.693,Z 287.555,A -85,B 0,C 180,E1 -27041.433,E2 -27041.433} C_VEL
LIN {X 0,Y 118.542,Z 301.152,A -85,B 0,C 180,E1 -27042.647,E2 -27042.647} C_VEL
LIN {X 0,Y 115.876,Z 312.932,A -85,B 0,C 180,E1 -27044.238,E2 -27044.238} C_VEL
LIN {X 0,Y 112.428,Z 324.934,A -85,B 0,C 180,E1 -27046.556,E2 -27046.556} C_VEL
LIN {X 0,Y 108.924,Z 335.142,A -85,B 0,C 180,E1 -27049.209,E2 -27049.209} C_VEL
LIN {X 0,Y 105.218,Z 344.662,A -85,B 0,C 180,E1 -27052.445,E2 -27052.445} C_VEL
LIN {X 0,Y 102.121,Z 352.35,A -85,B 0,C 180,E1 -27055.82,E2 -27055.82} C_VEL
LIN {X 0,Y 99.421,Z 358.607,A -85,B 0,C 180,E1 -27059.169,E2 -27059.169} C_VEL
LIN {X 0,Y 95.903,Z 367.134,A -85,B 0,C 180,E1 -27065.078,E2 -27065.078} C_VEL
LIN {X 0,Y 93.209,Z 373.942,A -85,B 0,C 180,E1 -27071.309,E2 -27071.309} C_VEL
LIN {X 0,Y 91.546,Z 380.173,A -85,B 0,C 180,E1 -27078.934,E2 -27078.934} C_VEL
LIN {X 0,Y 91.088,Z 384.172,A -85,B 0,C 180,E1 -27085.574,E2 -27085.574} C_VEL
LIN {X 0,Y 91.222,Z 386.206,A -85,B 0,C 180,E1 -27089.999,E2 -27089.999} C_VEL
LIN {X 0,Y 91.1,Z 387.767,A -85,B 0,C 180,E1 -27094.424,E2 -27094.424} C_VEL
LIN {X 0,Y 91.922,Z 389.684,A -85,B 0,C 180,E1 -27103.259,E2 -27103.259} C_VEL
LIN {X 0,Y 94.637,Z 390.004,A -85,B 0,C 180,E1 -27111.796,E2 -27111.796} C_VEL
LIN {X 0,Y 99.521,Z 388.853,A -85,B 0,C 180,E1 -27119.625,E2 -27119.625} C_VEL
LIN {X 0,Y 102.584,Z 387.692,A -85,B 0,C 180,E1 -27123.235,E2 -27123.235} C_VEL
LIN {X 0,Y 106.115,Z 386.113,A -85,B 0,C 180,E1 -27126.588,E2 -27126.588} C_VEL
LIN {X 0,Y 111.876,Z 382.993,A -85,B 0,C 180,E1 -27131.267,E2 -27131.267} C_VEL
LIN {X 0,Y 118.419,Z 378.859,A -85,B 0,C 180,E1 -27135.412,E2 -27135.412} C_VEL
LIN {X 0,Y 126.886,Z 372.587,A -85,B 0,C 180,E1 -27139.604,E2 -27139.604} C_VEL
LIN {X 0,Y 134.696,Z 365.796,A -85,B 0,C 180,E1 -27142.721,E2 -27142.721} C_VEL
LIN {X 0,Y 141.474,Z 358.905,A -85,B 0,C 180,E1 -27145.051,E2 -27145.051} C_VEL
LIN {X 0,Y 148.453,Z 350.672,A -85,B 0,C 180,E1 -27147.173,E2 -27147.173} C_VEL
LIN {X 0,Y 155.711,Z 340.608,A -85,B 0,C 180,E1 -27149.044,E2 -27149.044} C_VEL
LIN {X 0,Y 162.456,Z 329.25,A -85,B 0,C 180,E1 -27150.532,E2 -27150.532} C_VEL
LIN {X 0,Y 168.28,Z 316.964,A -85,B 0,C 180,E1 -27151.709,E2 -27151.709} C_VEL
LIN {X 0,Y 172.457,Z 305.531,A -85,B 0,C 180,E1 -27152.473,E2 -27152.473} C_VEL
LIN {X 0,Y 175.445,Z 294.505,A -85,B 0,C 180,E1 -27153.031,E2 -27153.031} C_VEL
LIN {X 0,Y 175.811,Z 291.57,A -85,B 0,C 180,E1 -27153.422,E2 -27153.422} C_VEL
LIN {X 0,Y 175.674,Z 288.655,A -85,B 0,C 180,E1 -27154.279,E2 -27154.279} C_VEL
LIN {X 0,Y 174.819,Z 285.394,A -85,B 0,C 180,E1 -27155.998,E2 -27155.998} C_VEL
LIN {X 0,Y 173.498,Z 281.676,A -85,B 0,C 180,E1 -27158.58,E2 -27158.58} C_VEL
LIN {X 0,Y 172.657,Z 278.71,A -85,B 0,C 180,E1 -27160.704,E2 -27160.704} C_VEL
LIN {X 0,Y 171.958,Z 276.275,A -85,B 0,C 180,E1 -27162.916,E2 -27162.916} C_VEL
LIN {X 0,Y 171.056,Z 273.269,A -85,B 0,C 180,E1 -27167.542,E2 -27167.542} C_VEL
LIN {X 0,Y 171.192,Z 273.255,A -85,B 0,C 180,E1 -27173.78,E2 -27173.78} C_VEL
LIN {X 0,Y 171.413,Z 273.943,A -85,B 0,C 180,E1 -27175.107,E2 -27175.107} C_VEL
LIN {X 0,Y 172.738,Z 277.418,A -85,B 0,C 180,E1 -27179.707,E2 -27179.707} C_VEL
LIN {X 0,Y 173.999,Z 280.805,A -85,B 0,C 180,E1 -27182.603,E2 -27182.603} C_VEL
LIN {X 0,Y 175.13,Z 283.996,A -85,B 0,C 180,E1 -27184.89,E2 -27184.89} C_VEL
LIN {X 0,Y 172.103,Z 297.384,A -85,B 0,C 180,E1 -27185.512,E2 -27185.512} C_VEL
LIN {X 0,Y 167.948,Z 309.834,A -85,B 0,C 180,E1 -27186.364,E2 -27186.364} C_VEL
LIN {X 0,Y 163.018,Z 321.137,A -85,B 0,C 180,E1 -27187.444,E2 -27187.444} C_VEL
LIN {X 0,Y 157.306,Z 331.53,A -85,B 0,C 180,E1 -27188.704,E2 -27188.704} C_VEL
LIN {X 0,Y 150.894,Z 341.193,A -85,B 0,C 180,E1 -27190.291,E2 -27190.291} C_VEL
LIN {X 0,Y 143.822,Z 350.062,A -85,B 0,C 180,E1 -27192.227,E2 -27192.227} C_VEL
LIN {X 0,Y 135.789,Z 358.499,A -85,B 0,C 180,E1 -27194.739,E2 -27194.739} C_VEL
LIN {X 0,Y 127.345,Z 365.933,A -85,B 0,C 180,E1 -27197.823,E2 -27197.823} C_VEL
LIN {X 0,Y 120.343,Z 371.144,A -85,B 0,C 180,E1 -27200.87,E2 -27200.87} C_VEL
LIN {X 0,Y 112.444,Z 376.109,A -85,B 0,C 180,E1 -27205.004,E2 -27205.004} C_VEL
LIN {X 0,Y 105.222,Z 379.817,A -85,B 0,C 180,E1 -27209.739,E2 -27209.739} C_VEL
LIN {X 0,Y 99.682,Z 382.051,A -85,B 0,C 180,E1 -27214.333,E2 -27214.333} C_VEL
LIN {X 0,Y 93.419,Z 383.836,A -85,B 0,C 180,E1 -27221.21,E2 -27221.21} C_VEL
LIN {X 0,Y 90.385,Z 384.221,A -85,B 0,C 180,E1 -27225.589,E2 -27225.589} C_VEL
LIN {X 0,Y 87.88,Z 384.17,A -85,B 0,C 180,E1 -27230.225,E2 -27230.225} C_VEL
LIN {X 0,Y 85.978,Z 383.69,A -85,B 0,C 180,E1 -27235.097,E2 -27235.097} C_VEL
LIN {X 0,Y 84.561,Z 382.723,A -85,B 0,C 180,E1 -27240.089,E2 -27240.089} C_VEL
LIN {X 0,Y 83.548,Z 380.464,A -85,B 0,C 180,E1 -27247.708,E2 -27247.708} C_VEL
LIN {X 0,Y 83.747,Z 377.107,A -85,B 0,C 180,E1 -27255.419,E2 -27255.419} C_VEL
LIN {X 0,Y 85.007,Z 372.713,A -85,B 0,C 180,E1 -27262.776,E2 -27262.776} C_VEL
LIN {X 0,Y 87.198,Z 366.956,A -85,B 0,C 180,E1 -27270.001,E2 -27270.001} C_VEL
LIN {X 0,Y 90.25,Z 359.879,A -85,B 0,C 180,E1 -27276.709,E2 -27276.709} C_VEL
LIN {X 0,Y 93.581,Z 352.749,A -85,B 0,C 180,E1 -27281.83,E2 -27281.83} C_VEL
LIN {X 0,Y 98.074,Z 342.822,A -85,B 0,C 180,E1 -27287.194,E2 -27287.194} C_VEL
LIN {X 0,Y 102.259,Z 332.931,A -85,B 0,C 180,E1 -27291.151,E2 -27291.151} C_VEL
LIN {X 0,Y 106.227,Z 322.125,A -85,B 0,C 180,E1 -27294.426,E2 -27294.426} C_VEL
LIN {X 0,Y 109.774,Z 310.556,A -85,B 0,C 180,E1 -27297.006,E2 -27297.006} C_VEL
LIN {X 0,Y 112.901,Z 297.697,A -85,B 0,C 180,E1 -27299.047,E2 -27299.047} C_VEL
LIN {X 0,Y 115.114,Z 284.727,A -85,B 0,C 180,E1 -27300.458,E2 -27300.458} C_VEL
LIN {X 0,Y 116.768,Z 268.743,A -85,B 0,C 180,E1 -27301.406,E2 -27301.406} C_VEL
LIN {X 0,Y 119.133,Z 239.082,A -85,B 0,C 180,E1 -27302.855,E2 -27302.855} C_VEL
LIN {X 0,Y 115.068,Z 229.717,A -85,B 0,C 180,E1 -27305.757,E2 -27305.757} C_VEL
LIN {X 0,Y 110.789,Z 221.393,A -85,B 0,C 180,E1 -27309.089,E2 -27309.089} C_VEL
LIN {X 0,Y 106.311,Z 213.827,A -85,B 0,C 180,E1 -27313.006,E2 -27313.006} C_VEL
LIN {X 0,Y 102.401,Z 208.037,A -85,B 0,C 180,E1 -27316.929,E2 -27316.929} C_VEL
LIN {X 0,Y 99.821,Z 204.345,A -85,B 0,C 180,E1 -27319.946,E2 -27319.946} C_VEL
LIN {X 0,Y 96.974,Z 200.872,A -85,B 0,C 180,E1 -27323.767,E2 -27323.767} C_VEL
LIN {X 0,Y 96.163,Z 199.227,A -85,B 0,C 180,E1 -27325.123,E2 -27325.123} C_VEL
LIN {X 0,Y 93.158,Z 196.571,A -85,B 0,C 180,E1 -27330.327,E2 -27330.327} C_VEL
LIN {X 0,Y 91.825,Z 193.653,A -85,B 0,C 180,E1 -27333.755,E2 -27333.755} C_VEL
LIN {X 0,Y 88.682,Z 191.472,A -85,B 0,C 180,E1 -27348.575,E2 -27348.575} C_VEL
LIN {X 0,Y 89.459,Z 191.798,A -85,B 0,C 180,E1 -27357.751,E2 -27357.751} C_VEL
LIN {X 0,Y 90.122,Z 192.161,A -85,B 0,C 180,E1 -27360.561,E2 -27360.561} C_VEL
LIN {X 0,Y 92.406,Z 193.738,A -85,B 0,C 180,E1 -27366.963,E2 -27366.963} C_VEL
LIN {X 0,Y 93.637,Z 196.556,A -85,B 0,C 180,E1 -27369.971,E2 -27369.971} C_VEL
LIN {X 0,Y 96.013,Z 198.965,A -85,B 0,C 180,E1 -27374.102,E2 -27374.102} C_VEL
LIN {X 0,Y 96.541,Z 199.707,A -85,B 0,C 180,E1 -27374.949,E2 -27374.949} C_VEL
LIN {X 0,Y 98.585,Z 202.917,A -85,B 0,C 180,E1 -27377.974,E2 -27377.974} C_VEL
LIN {X 0,Y 100.041,Z 204.5,A -85,B 0,C 180,E1 -27379.779,E2 -27379.779} C_VEL
LIN {X 0,Y 102.728,Z 208.278,A -85,B 0,C 180,E1 -27382.865,E2 -27382.865} C_VEL
LIN {X 0,Y 106.644,Z 214.383,A -85,B 0,C 180,E1 -27386.778,E2 -27386.778} C_VEL
LIN {X 0,Y 111.345,Z 222.496,A -85,B 0,C 180,E1 -27390.856,E2 -27390.856} C_VEL
LIN {X 0,Y 113.696,Z 227.469,A -85,B 0,C 180,E1 -27392.745,E2 -27392.745} C_VEL
LIN {X 0,Y 117.141,Z 237.796,A -85,B 0,C 180,E1 -27395.538,E2 -27395.538} C_VEL
LIN {X 0,Y 118.406,Z 242.203,A -85,B 0,C 180,E1 -27396.544,E2 -27396.544} C_VEL
LIN {X 0,Y 118.609,Z 248.923,A -85,B 0,C 180,E1 -27397.219,E2 -27397.219} C_VEL
LIN {X 0,Y 115.382,Z 287.009,A -85,B 0,C 180,E1 -27399.149,E2 -27399.149} C_VEL
LIN {X 0,Y 113.141,Z 300.671,A -85,B 0,C 180,E1 -27400.373,E2 -27400.373} C_VEL
LIN {X 0,Y 110.137,Z 313.281,A -85,B 0,C 180,E1 -27402.113,E2 -27402.113} C_VEL
LIN {X 0,Y 106.819,Z 324.352,A -85,B 0,C 180,E1 -27404.314,E2 -27404.314} C_VEL
LIN {X 0,Y 103.072,Z 334.601,A -85,B 0,C 180,E1 -27407.01,E2 -27407.01} C_VEL
LIN {X 0,Y 99.151,Z 344.173,A -85,B 0,C 180,E1 -27410.361,E2 -27410.361} C_VEL
LIN {X 0,Y 95.739,Z 352.179,A -85,B 0,C 180,E1 -27414.036,E2 -27414.036} C_VEL
LIN {X 0,Y 92.628,Z 358.974,A -85,B 0,C 180,E1 -27417.918,E2 -27417.918} C_VEL
LIN {X 0,Y 88.895,Z 367.369,A -85,B 0,C 180,E1 -27424.225,E2 -27424.225} C_VEL
LIN {X 0,Y 86.116,Z 374.09,A -85,B 0,C 180,E1 -27430.946,E2 -27430.946} C_VEL
LIN {X 0,Y 84.546,Z 379.432,A -85,B 0,C 180,E1 -27438.005,E2 -27438.005} C_VEL
LIN {X 0,Y 84.004,Z 383.546,A -85,B 0,C 180,E1 -27445.2,E2 -27445.2} C_VEL
LIN {X 0,Y 84.138,Z 385.676,A -85,B 0,C 180,E1 -27449.999,E2 -27449.999} C_VEL
LIN {X 0,Y 84.033,Z 387.287,A -85,B 0,C 180,E1 -27454.797,E2 -27454.797} C_VEL
LIN {X 0,Y 85.001,Z 389.311,A -85,B 0,C 180,E1 -27464.361,E2 -27464.361} C_VEL
LIN {X 0,Y 86.262,Z 389.743,A -85,B 0,C 180,E1 -27469.019,E2 -27469.019} C_VEL
LIN {X 0,Y 90.487,Z 389.426,A -85,B 0,C 180,E1 -27477.775,E2 -27477.775} C_VEL
LIN {X 0,Y 96.713,Z 387.628,A -85,B 0,C 180,E1 -27485.545,E2 -27485.545} C_VEL
LIN {X 0,Y 100.484,Z 386.122,A -85,B 0,C 180,E1 -27489.011,E2 -27489.011} C_VEL
LIN {X 0,Y 106.637,Z 383.105,A -85,B 0,C 180,E1 -27493.786,E2 -27493.786} C_VEL
LIN {X 0,Y 113.552,Z 379.076,A -85,B 0,C 180,E1 -27497.962,E2 -27497.962} C_VEL
LIN {X 0,Y 122.422,Z 372.949,A -85,B 0,C 180,E1 -27502.125,E2 -27502.125} C_VEL
LIN {X 0,Y 130.536,Z 366.312,A -85,B 0,C 180,E1 -27505.19,E2 -27505.19} C_VEL
LIN {X 0,Y 138.982,Z 358.122,A -85,B 0,C 180,E1 -27507.887,E2 -27507.887} C_VEL
LIN {X 0,Y 146.232,Z 349.781,A -85,B 0,C 180,E1 -27509.893,E2 -27509.893} C_VEL
LIN {X 0,Y 153.734,Z 339.518,A -85,B 0,C 180,E1 -27511.644,E2 -27511.644} C_VEL
LIN {X 0,Y 160.656,Z 327.986,A -85,B 0,C 180,E1 -27513.039,E2 -27513.039} C_VEL
LIN {X 0,Y 166.323,Z 316.092,A -85,B 0,C 180,E1 -27514.081,E2 -27514.081} C_VEL
LIN {X 0,Y 170.851,Z 303.655,A -85,B 0,C 180,E1 -27514.82,E2 -27514.82} C_VEL
LIN {X 0,Y 174.335,Z 290.005,A -85,B 0,C 180,E1 -27515.426,E2 -27515.426} C_VEL
LIN {X 0,Y 174.792,Z 287.174,A -85,B 0,C 180,E1 -27515.582,E2 -27515.582} C_VEL
LIN {X 0,Y 173.617,Z 282.048,A -85,B 0,C 180,E1 -27518.322,E2 -27518.322} C_VEL
LIN {X 0,Y 173.498,Z 281.676,A -85,B 0,C 180,E1 -27518.58,E2 -27518.58} C_VEL
LIN {X 0,Y 172.966,Z 280.219,A -85,B 0,C 180,E1 -27519.772,E2 -27519.772} C_VEL
LIN {X 0,Y 172.098,Z 279.204,A -85,B 0,C 180,E1 -27521.686,E2 -27521.686} C_VEL
LIN {X 0,Y 170.785,Z 279.462,A -85,B 0,C 180,E1 -27525.018,E2 -27525.018} C_VEL
LIN {X 0,Y 169.918,Z 280.211,A -85,B 0,C 180,E1 -27529.135,E2 -27529.135} C_VEL
LIN {X 0,Y 170.203,Z 280.286,A -85,B 0,C 180,E1 -27533.744,E2 -27533.744} C_VEL
LIN {X 0,Y 171.291,Z 284.163,A -85,B 0,C 180,E1 -27539.117,E2 -27539.117} C_VEL
LIN {X 0,Y 172.181,Z 287.374,A -85,B 0,C 180,E1 -27541.899,E2 -27541.899} C_VEL
LIN {X 0,Y 172.52,Z 288.483,A -85,B 0,C 180,E1 -27542.808,E2 -27542.808} C_VEL
LIN {X 0,Y 168.978,Z 301.735,A -85,B 0,C 180,E1 -27543.45,E2 -27543.45} C_VEL
LIN {X 0,Y 164.615,Z 313.492,A -85,B 0,C 180,E1 -27544.286,E2 -27544.286} C_VEL
LIN {X 0,Y 159.146,Z 324.803,A -85,B 0,C 180,E1 -27545.394,E2 -27545.394} C_VEL
LIN {X 0,Y 152.189,Z 336.216,A -85,B 0,C 180,E1 -27546.851,E2 -27546.851} C_VEL
LIN {X 0,Y 144.439,Z 346.537,A -85,B 0,C 180,E1 -27548.701,E2 -27548.701} C_VEL
LIN {X 0,Y 136.027,Z 355.718,A -85,B 0,C 180,E1 -27550.992,E2 -27550.992} C_VEL
LIN {X 0,Y 126.726,Z 364.11,A -85,B 0,C 180,E1 -27553.947,E2 -27553.947} C_VEL
LIN {X 0,Y 117.821,Z 370.676,A -85,B 0,C 180,E1 -27557.371,E2 -27557.371} C_VEL
LIN {X 0,Y 109.417,Z 375.8,A -85,B 0,C 180,E1 -27561.354,E2 -27561.354} C_VEL
LIN {X 0,Y 101.617,Z 379.65,A -85,B 0,C 180,E1 -27565.961,E2 -27565.961} C_VEL
LIN {X 0,Y 94.592,Z 382.346,A -85,B 0,C 180,E1 -27571.335,E2 -27571.335} C_VEL
LIN {X 0,Y 88.529,Z 383.947,A -85,B 0,C 180,E1 -27577.453,E2 -27577.453} C_VEL
LIN {X 0,Y 85.06,Z 384.463,A -85,B 0,C 180,E1 -27581.961,E2 -27581.961} C_VEL
LIN {X 0,Y 82.124,Z 384.484,A -85,B 0,C 180,E1 -27586.795,E2 -27586.795} C_VEL
LIN {X 0,Y 79.51,Z 383.993,A -85,B 0,C 180,E1 -27592.7,E2 -27592.7} C_VEL
LIN {X 0,Y 78.06,Z 383.237,A -85,B 0,C 180,E1 -27597.304,E2 -27597.304} C_VEL
LIN {X 0,Y 76.514,Z 380.725,A -85,B 0,C 180,E1 -27606.704,E2 -27606.704} C_VEL
LIN {X 0,Y 76.788,Z 376.577,A -85,B 0,C 180,E1 -27616.774,E2 -27616.774} C_VEL
LIN {X 0,Y 78.316,Z 371.886,A -85,B 0,C 180,E1 -27624.852,E2 -27624.852} C_VEL
LIN {X 0,Y 80.799,Z 365.947,A -85,B 0,C 180,E1 -27632.494,E2 -27632.494} C_VEL
LIN {X 0,Y 84.405,Z 358.48,A -85,B 0,C 180,E1 -27639.587,E2 -27639.587} C_VEL
LIN {X 0,Y 89.036,Z 349.204,A -85,B 0,C 180,E1 -27646.039,E2 -27646.039} C_VEL
LIN {X 0,Y 93.597,Z 339.571,A -85,B 0,C 180,E1 -27650.897,E2 -27650.897} C_VEL
LIN {X 0,Y 98.107,Z 328.861,A -85,B 0,C 180,E1 -27654.89,E2 -27654.89} C_VEL
LIN {X 0,Y 102.518,Z 316.876,A -85,B 0,C 180,E1 -27658.12,E2 -27658.12} C_VEL
LIN {X 0,Y 106.104,Z 304.29,A -85,B 0,C 180,E1 -27660.567,E2 -27660.567} C_VEL
LIN {X 0,Y 109.015,Z 290.871,A -85,B 0,C 180,E1 -27662.352,E2 -27662.352} C_VEL
LIN {X 0,Y 110.875,Z 277.828,A -85,B 0,C 180,E1 -27663.409,E2 -27663.409} C_VEL
LIN {X 0,Y 113.999,Z 241.244,A -85,B 0,C 180,E1 -27665.249,E2 -27665.249} C_VEL
LIN {X 0,Y 109.688,Z 231.407,A -85,B 0,C 180,E1 -27668.736,E2 -27668.736} C_VEL
LIN {X 0,Y 105.703,Z 223.687,A -85,B 0,C 180,E1 -27672.3,E2 -27672.3} C_VEL
LIN {X 0,Y 102.047,Z 217.51,A -85,B 0,C 180,E1 -27675.972,E2 -27675.972} C_VEL
LIN {X 0,Y 99.48,Z 213.648,A -85,B 0,C 180,E1 -27678.898,E2 -27678.898} C_VEL
LIN {X 0,Y 96.943,Z 209.895,A -85,B 0,C 180,E1 -27682.238,E2 -27682.238} C_VEL
LIN {X 0,Y 94.607,Z 206.591,A -85,B 0,C 180,E1 -27685.859,E2 -27685.859} C_VEL
LIN {X 0,Y 93.941,Z 205.603,A -85,B 0,C 180,E1 -27687.032,E2 -27687.032} C_VEL
LIN {X 0,Y 91.233,Z 202.584,A -85,B 0,C 180,E1 -27692.474,E2 -27692.474} C_VEL
LIN {X 0,Y 90.387,Z 200.556,A -85,B 0,C 180,E1 -27694.979,E2 -27694.979} C_VEL
LIN {X 0,Y 87.777,Z 198.503,A -85,B 0,C 180,E1 -27708.864,E2 -27708.864} C_VEL
LIN {X 0,Y 88.925,Z 198.966,A -85,B 0,C 180,E1 -27719.436,E2 -27719.436} C_VEL
LIN {X 0,Y 90.865,Z 200.597,A -85,B 0,C 180,E1 -27725.613,E2 -27725.613} C_VEL
LIN {X 0,Y 92.498,Z 203.821,A -85,B 0,C 180,E1 -27729.7,E2 -27729.7} C_VEL
LIN {X 0,Y 94.458,Z 205.966,A -85,B 0,C 180,E1 -27733.288,E2 -27733.288} C_VEL
LIN {X 0,Y 96.707,Z 209.543,A -85,B 0,C 180,E1 -27736.902,E2 -27736.902} C_VEL
LIN {X 0,Y 97.784,Z 210.898,A -85,B 0,C 180,E1 -27738.369,E2 -27738.369} C_VEL
LIN {X 0,Y 101.115,Z 216.031,A -85,B 0,C 180,E1 -27742.471,E2 -27742.471} C_VEL
LIN {X 0,Y 104.445,Z 221.501,A -85,B 0,C 180,E1 -27745.963,E2 -27745.963} C_VEL
LIN {X 0,Y 108.948,Z 229.954,A -85,B 0,C 180,E1 -27750.118,E2 -27750.118} C_VEL
LIN {X 0,Y 112.201,Z 239.868,A -85,B 0,C 180,E1 -27753.103,E2 -27753.103} C_VEL
LIN {X 0,Y 113.465,Z 244.893,A -85,B 0,C 180,E1 -27754.284,E2 -27754.284} C_VEL
LIN {X 0,Y 113.525,Z 249.829,A -85,B 0,C 180,E1 -27754.779,E2 -27754.779} C_VEL
LIN {X 0,Y 110.236,Z 286.719,A -85,B 0,C 180,E1 -27756.666,E2 -27756.666} C_VEL
LIN {X 0,Y 107.789,Z 300.883,A -85,B 0,C 180,E1 -27757.951,E2 -27757.951} C_VEL
LIN {X 0,Y 104.881,Z 312.596,A -85,B 0,C 180,E1 -27759.59,E2 -27759.59} C_VEL
LIN {X 0,Y 101.376,Z 323.762,A -85,B 0,C 180,E1 -27761.818,E2 -27761.818} C_VEL
LIN {X 0,Y 97.408,Z 334.068,A -85,B 0,C 180,E1 -27764.561,E2 -27764.561} C_VEL
LIN {X 0,Y 93.25,Z 343.69,A -85,B 0,C 180,E1 -27768.018,E2 -27768.018} C_VEL
LIN {X 0,Y 89.379,Z 352.12,A -85,B 0,C 180,E1 -27772.051,E2 -27772.051} C_VEL
LIN {X 0,Y 85.87,Z 359.313,A -85,B 0,C 180,E1 -27776.463,E2 -27776.463} C_VEL
LIN {X 0,Y 81.899,Z 367.602,A -85,B 0,C 180,E1 -27783.222,E2 -27783.222} C_VEL
LIN {X 0,Y 79.383,Z 373.212,A -85,B 0,C 180,E1 -27789.259,E2 -27789.259} C_VEL
LIN {X 0,Y 77.588,Z 378.68,A -85,B 0,C 180,E1 -27796.911,E2 -27796.911} C_VEL
LIN {X 0,Y 76.92,Z 382.91,A -85,B 0,C 180,E1 -27804.757,E2 -27804.757} C_VEL
LIN {X 0,Y 77.056,Z 385.128,A -85,B 0,C 180,E1 -27809.999,E2 -27809.999} C_VEL
LIN {X 0,Y 76.961,Z 386.807,A -85,B 0,C 180,E1 -27815.239,E2 -27815.239} C_VEL
LIN {X 0,Y 78.127,Z 388.929,A -85,B 0,C 180,E1 -27825.656,E2 -27825.656} C_VEL
LIN {X 0,Y 81.567,Z 389.53,A -85,B 0,C 180,E1 -27835.518,E2 -27835.518} C_VEL
LIN {X 0,Y 87.413,Z 388.574,A -85,B 0,C 180,E1 -27844.249,E2 -27844.249} C_VEL
LIN {X 0,Y 95.057,Z 386.122,A -85,B 0,C 180,E1 -27851.713,E2 -27851.713} C_VEL
LIN {X 0,Y 101.624,Z 383.192,A -85,B 0,C 180,E1 -27856.564,E2 -27856.564} C_VEL
LIN {X 0,Y 108.923,Z 379.279,A -85,B 0,C 180,E1 -27860.739,E2 -27860.739} C_VEL
LIN {X 0,Y 116.835,Z 374.279,A -85,B 0,C 180,E1 -27864.298,E2 -27864.298} C_VEL
LIN {X 0,Y 125.231,Z 368.036,A -85,B 0,C 180,E1 -27867.331,E2 -27867.331} C_VEL
LIN {X 0,Y 133.887,Z 360.289,A -85,B 0,C 180,E1 -27870.01,E2 -27870.01} C_VEL
LIN {X 0,Y 141.312,Z 352.43,A -85,B 0,C 180,E1 -27871.979,E2 -27871.979} C_VEL
LIN {X 0,Y 149.742,Z 341.803,A -85,B 0,C 180,E1 -27873.846,E2 -27873.846} C_VEL
LIN {X 0,Y 156.81,Z 330.947,A -85,B 0,C 180,E1 -27875.173,E2 -27875.173} C_VEL
LIN {X 0,Y 162.921,Z 319.156,A -85,B 0,C 180,E1 -27876.207,E2 -27876.207} C_VEL
LIN {X 0,Y 167.42,Z 308.116,A -85,B 0,C 180,E1 -27876.914,E2 -27876.914} C_VEL
LIN {X 0,Y 171.406,Z 294.956,A -85,B 0,C 180,E1 -27877.518,E2 -27877.518} C_VEL
LIN {X 0,Y 172.272,Z 290.959,A -85,B 0,C 180,E1 -27877.71,E2 -27877.71} C_VEL
LIN {X 0,Y 171.413,Z 286.219,A -85,B 0,C 180,E1 -27880.653,E2 -27880.653} C_VEL
LIN {X 0,Y 170.725,Z 283.017,A -85,B 0,C 180,E1 -27883.559,E2 -27883.559} C_VEL
LIN {X 0,Y 170.09,Z 280.388,A -85,B 0,C 180,E1 -27887.47,E2 -27887.47} C_VEL
LIN {X 0,Y 169.918,Z 280.211,A -85,B 0,C 180,E1 -27889.135,E2 -27889.135} C_VEL
LIN {X 0,Y 169.83,Z 280.535,A -85,B 0,C 180,E1 -27890.455,E2 -27890.455} C_VEL
LIN {X 0,Y 169.737,Z 281.507,A -85,B 0,C 180,E1 -27891.744,E2 -27891.744} C_VEL
LIN {X 0,Y 169.519,Z 284.661,A -85,B 0,C 180,E1 -27894.212,E2 -27894.212} C_VEL
LIN {X 0,Y 169.442,Z 290.133,A -85,B 0,C 180,E1 -27897.905,E2 -27897.905} C_VEL
LIN {X 0,Y 169.656,Z 291.497,A -85,B 0,C 180,E1 -27899.194,E2 -27899.194} C_VEL
LIN {X 0,Y 169.946,Z 293.166,A -85,B 0,C 180,E1 -27900.65,E2 -27900.65} C_VEL
LIN {X 0,Y 165.855,Z 306.319,A -85,B 0,C 180,E1 -27901.348,E2 -27901.348} C_VEL
LIN {X 0,Y 160.915,Z 318.122,A -85,B 0,C 180,E1 -27902.255,E2 -27902.255} C_VEL
LIN {X 0,Y 154.881,Z 329.259,A -85,B 0,C 180,E1 -27903.351,E2 -27903.351} C_VEL
LIN {X 0,Y 148.085,Z 339.39,A -85,B 0,C 180,E1 -27904.694,E2 -27904.694} C_VEL
LIN {X 0,Y 139.721,Z 349.634,A -85,B 0,C 180,E1 -27906.571,E2 -27906.571} C_VEL
LIN {X 0,Y 131.527,Z 357.904,A -85,B 0,C 180,E1 -27908.697,E2 -27908.697} C_VEL
LIN {X 0,Y 121.947,Z 365.833,A -85,B 0,C 180,E1 -27911.555,E2 -27911.555} C_VEL
LIN {X 0,Y 112.167,Z 372.482,A -85,B 0,C 180,E1 -27915.171,E2 -27915.171} C_VEL
LIN {X 0,Y 104.003,Z 376.983,A -85,B 0,C 180,E1 -27918.907,E2 -27918.907} C_VEL
LIN {X 0,Y 95.853,Z 380.581,A -85,B 0,C 180,E1 -27923.581,E2 -27923.581} C_VEL
LIN {X 0,Y 88.458,Z 383.037,A -85,B 0,C 180,E1 -27929.08,E2 -27929.08} C_VEL
LIN {X 0,Y 84.048,Z 384.063,A -85,B 0,C 180,E1 -27933.261,E2 -27933.261} C_VEL
LIN {X 0,Y 80.066,Z 384.662,A -85,B 0,C 180,E1 -27937.908,E2 -27937.908} C_VEL
LIN {X 0,Y 76.689,Z 384.798,A -85,B 0,C 180,E1 -27942.85,E2 -27942.85} C_VEL
LIN {X 0,Y 73.031,Z 384.248,A -85,B 0,C 180,E1 -27950.337,E2 -27950.337} C_VEL
LIN {X 0,Y 70.243,Z 382.491,A -85,B 0,C 180,E1 -27959.983,E2 -27959.983} C_VEL
LIN {X 0,Y 69.303,Z 379.792,A -85,B 0,C 180,E1 -27969.211,E2 -27969.211} C_VEL
LIN {X 0,Y 69.877,Z 376.001,A -85,B 0,C 180,E1 -27978.396,E2 -27978.396} C_VEL
LIN {X 0,Y 71.691,Z 371.051,A -85,B 0,C 180,E1 -27987.191,E2 -27987.191} C_VEL
LIN {X 0,Y 74.697,Z 364.803,A -85,B 0,C 180,E1 -27995.4,E2 -27995.4} C_VEL
LIN {X 0,Y 78.745,Z 357.055,A -85,B 0,C 180,E1 -28002.896,E2 -28002.896} C_VEL
LIN {X 0,Y 82.983,Z 349.121,A -85,B 0,C 180,E1 -28008.519,E2 -28008.519} C_VEL
LIN {X 0,Y 87.891,Z 339.386,A -85,B 0,C 180,E1 -28013.568,E2 -28013.568} C_VEL
LIN {X 0,Y 92.704,Z 328.587,A -85,B 0,C 180,E1 -28017.669,E2 -28017.669} C_VEL
LIN {X 0,Y 96.782,Z 318.128,A -85,B 0,C 180,E1 -28020.553,E2 -28020.553} C_VEL
LIN {X 0,Y 100.687,Z 305.468,A -85,B 0,C 180,E1 -28023.116,E2 -28023.116} C_VEL
LIN {X 0,Y 103.822,Z 292.172,A -85,B 0,C 180,E1 -28024.922,E2 -28024.922} C_VEL
LIN {X 0,Y 105.728,Z 279.982,A -85,B 0,C 180,E1 -28026.017,E2 -28026.017} C_VEL
LIN {X 0,Y 109.064,Z 243.521,A -85,B 0,C 180,E1 -28027.864,E2 -28027.864} C_VEL
LIN {X 0,Y 104.829,Z 233.705,A -85,B 0,C 180,E1 -28031.772,E2 -28031.772} C_VEL
LIN {X 0,Y 100.635,Z 225.685,A -85,B 0,C 180,E1 -28036.118,E2 -28036.118} C_VEL
LIN {X 0,Y 97.134,Z 219.873,A -85,B 0,C 180,E1 -28040.389,E2 -28040.389} C_VEL
LIN {X 0,Y 94.725,Z 216.114,A -85,B 0,C 180,E1 -28043.884,E2 -28043.884} C_VEL
LIN {X 0,Y 92.034,Z 212.051,A -85,B 0,C 180,E1 -28048.656,E2 -28048.656} C_VEL
LIN {X 0,Y 89.645,Z 209.035,A -85,B 0,C 180,E1 -28054.06,E2 -28054.06} C_VEL
LIN {X 0,Y 89.002,Z 207.452,A -85,B 0,C 180,E1 -28056.205,E2 -28056.205} C_VEL
LIN {X 0,Y 86.879,Z 205.558,A -85,B 0,C 180,E1 -28068.747,E2 -28068.747} C_VEL
LIN {X 0,Y 87.416,Z 205.781,A -85,B 0,C 180,E1 -28076.546,E2 -28076.546} C_VEL
LIN {X 0,Y 88.449,Z 206.61,A -85,B 0,C 180,E1 -28081.283,E2 -28081.283} C_VEL
LIN {X 0,Y 89.47,Z 207.568,A -85,B 0,C 180,E1 -28084.508,E2 -28084.508} C_VEL
LIN {X 0,Y 91.329,Z 210.974,A -85,B 0,C 180,E1 -28089.34,E2 -28089.34} C_VEL
LIN {X 0,Y 92.613,Z 212.583,A -85,B 0,C 180,E1 -28091.88,E2 -28091.88} C_VEL
LIN {X 0,Y 94.97,Z 216.271,A -85,B 0,C 180,E1 -28095.942,E2 -28095.942} C_VEL
LIN {X 0,Y 98.263,Z 221.562,A -85,B 0,C 180,E1 -28100.53,E2 -28100.53} C_VEL
LIN {X 0,Y 101.771,Z 227.817,A -85,B 0,C 180,E1 -28104.609,E2 -28104.609} C_VEL
LIN {X 0,Y 105.364,Z 235.053,A -85,B 0,C 180,E1 -28108.237,E2 -28108.237} C_VEL
LIN {X 0,Y 108.183,Z 244.816,A -85,B 0,C 180,E1 -28111.205,E2 -28111.205} C_VEL
LIN {X 0,Y 108.734,Z 247.75,A -85,B 0,C 180,E1 -28111.852,E2 -28111.852} C_VEL
LIN {X 0,Y 108.328,Z 254.305,A -85,B 0,C 180,E1 -28112.281,E2 -28112.281} C_VEL
LIN {X 0,Y 105.248,Z 286.955,A -85,B 0,C 180,E1 -28113.99,E2 -28113.99} C_VEL
LIN {X 0,Y 102.726,Z 300.74,A -85,B 0,C 180,E1 -28115.242,E2 -28115.242} C_VEL
LIN {X 0,Y 99.531,Z 312.94,A -85,B 0,C 180,E1 -28116.984,E2 -28116.984} C_VEL
LIN {X 0,Y 95.556,Z 324.775,A -85,B 0,C 180,E1 -28119.441,E2 -28119.441} C_VEL
LIN {X 0,Y 91.413,Z 334.856,A -85,B 0,C 180,E1 -28122.268,E2 -28122.268} C_VEL
LIN {X 0,Y 87.02,Z 344.294,A -85,B 0,C 180,E1 -28125.845,E2 -28125.845} C_VEL
LIN {X 0,Y 83.822,Z 350.915,A -85,B 0,C 180,E1 -28129.143,E2 -28129.143} C_VEL
LIN {X 0,Y 79.982,Z 358.133,A -85,B 0,C 180,E1 -28133.62,E2 -28133.62} C_VEL
LIN {X 0,Y 75.601,Z 366.591,A -85,B 0,C 180,E1 -28140.786,E2 -28140.786} C_VEL
LIN {X 0,Y 72.303,Z 373.358,A -85,B 0,C 180,E1 -28148.621,E2 -28148.621} C_VEL
LIN {X 0,Y 70.274,Z 379.533,A -85,B 0,C 180,E1 -28158.461,E2 -28158.461} C_VEL
LIN {X 0,Y 69.832,Z 383.488,A -85,B 0,C 180,E1 -28167.115,E2 -28167.115} C_VEL
LIN {X 0,Y 69.961,Z 384.547,A -85,B 0,C 180,E1 -28169.999,E2 -28169.999} C_VEL
LIN {X 0,Y 69.914,Z 386.322,A -85,B 0,C 180,E1 -28175.768,E2 -28175.768} C_VEL
LIN {X 0,Y 71.31,Z 388.547,A -85,B 0,C 180,E1 -28187.197,E2 -28187.197} C_VEL
LIN {X 0,Y 75.197,Z 389.261,A -85,B 0,C 180,E1 -28197.859,E2 -28197.859} C_VEL
LIN {X 0,Y 78.158,Z 389.051,A -85,B 0,C 180,E1 -28202.65,E2 -28202.65} C_VEL
LIN {X 0,Y 85.545,Z 387.458,A -85,B 0,C 180,E1 -28211.089,E2 -28211.089} C_VEL
LIN {X 0,Y 94.459,Z 384.344,A -85,B 0,C 180,E1 -28218.075,E2 -28218.075} C_VEL
LIN {X 0,Y 101.938,Z 380.879,A -85,B 0,C 180,E1 -28222.453,E2 -28222.453} C_VEL
LIN {X 0,Y 110.052,Z 376.373,A -85,B 0,C 180,E1 -28226.117,E2 -28226.117} C_VEL
LIN {X 0,Y 120.075,Z 369.607,A -85,B 0,C 180,E1 -28229.691,E2 -28229.691} C_VEL
LIN {X 0,Y 128.975,Z 362.303,A -85,B 0,C 180,E1 -28232.311,E2 -28232.311} C_VEL
LIN {X 0,Y 138.142,Z 353.287,A -85,B 0,C 180,E1 -28234.56,E2 -28234.56} C_VEL
LIN {X 0,Y 146.774,Z 342.908,A -85,B 0,C 180,E1 -28236.314,E2 -28236.314} C_VEL
LIN {X 0,Y 153.99,Z 332.368,A -85,B 0,C 180,E1 -28237.547,E2 -28237.547} C_VEL
LIN {X 0,Y 160.325,Z 320.901,A -85,B 0,C 180,E1 -28238.524,E2 -28238.524} C_VEL
LIN {X 0,Y 165.361,Z 309.182,A -85,B 0,C 180,E1 -28239.231,E2 -28239.231} C_VEL
LIN {X 0,Y 169.716,Z 295.424,A -85,B 0,C 180,E1 -28239.824,E2 -28239.824} C_VEL
LIN {X 0,Y 169.775,Z 294.785,A -85,B 0,C 180,E1 -28240.029,E2 -28240.029} C_VEL
LIN {X 0,Y 169.435,Z 291.926,A -85,B 0,C 180,E1 -28242.09,E2 -28242.09} C_VEL
LIN {X 0,Y 169.179,Z 289.808,A -85,B 0,C 180,E1 -28244.024,E2 -28244.024} C_VEL
LIN {X 0,Y 168.769,Z 287.266,A -85,B 0,C 180,E1 -28247.981,E2 -28247.981} C_VEL
LIN {X 0,Y 168.902,Z 287.27,A -85,B 0,C 180,E1 -28253.696,E2 -28253.696} C_VEL
LIN {X 0,Y 169.519,Z 290.815,A -85,B 0,C 180,E1 -28258.514,E2 -28258.514} C_VEL
LIN {X 0,Y 169.656,Z 291.497,A -85,B 0,C 180,E1 -28259.194,E2 -28259.194} C_VEL
LIN {X 0,Y 169.598,Z 292.706,A -85,B 0,C 180,E1 -28259.716,E2 -28259.716} C_VEL
LIN {X 0,Y 169.042,Z 295.143,A -85,B 0,C 180,E1 -28260.039,E2 -28260.039} C_VEL
LIN {X 0,Y 167.845,Z 299.01,A -85,B 0,C 180,E1 -28260.03,E2 -28260.03} C_VEL
LIN {X 0,Y 163.803,Z 308.817,A -85,B 0,C 180,E1 -28259.221,E2 -28259.221} C_VEL
LIN {X 0,Y 162.58,Z 311.586,A -85,B 0,C 180,E1 -28259.251,E2 -28259.251} C_VEL
LIN {X 0,Y 156.972,Z 323.28,A -85,B 0,C 180,E1 -28260.175,E2 -28260.175} C_VEL
LIN {X 0,Y 150.261,Z 334.237,A -85,B 0,C 180,E1 -28261.284,E2 -28261.284} C_VEL
LIN {X 0,Y 142.17,Z 344.911,A -85,B 0,C 180,E1 -28262.832,E2 -28262.832} C_VEL
LIN {X 0,Y 133.957,Z 353.798,A -85,B 0,C 180,E1 -28264.567,E2 -28264.567} C_VEL
LIN {X 0,Y 125.853,Z 361.138,A -85,B 0,C 180,E1 -28266.576,E2 -28266.576} C_VEL
LIN {X 0,Y 115.794,Z 368.617,A -85,B 0,C 180,E1 -28269.505,E2 -28269.505} C_VEL
LIN {X 0,Y 107.88,Z 373.482,A -85,B 0,C 180,E1 -28272.26,E2 -28272.26} C_VEL
LIN {X 0,Y 97.665,Z 378.556,A -85,B 0,C 180,E1 -28276.726,E2 -28276.726} C_VEL
LIN {X 0,Y 90.266,Z 381.419,A -85,B 0,C 180,E1 -28280.885,E2 -28280.885} C_VEL
LIN {X 0,Y 84.971,Z 383.047,A -85,B 0,C 180,E1 -28284.522,E2 -28284.522} C_VEL
LIN {X 0,Y 80.066,Z 384.178,A -85,B 0,C 180,E1 -28288.625,E2 -28288.625} C_VEL
LIN {X 0,Y 74.601,Z 384.948,A -85,B 0,C 180,E1 -28294.416,E2 -28294.416} C_VEL
LIN {X 0,Y 68.327,Z 384.839,A -85,B 0,C 180,E1 -28303.946,E2 -28303.946} C_VEL
LIN {X 0,Y 65.697,Z 384.139,A -85,B 0,C 180,E1 -28310.071,E2 -28310.071} C_VEL
LIN {X 0,Y 63.77,Z 383.018,A -85,B 0,C 180,E1 -28316.563,E2 -28316.563} C_VEL
LIN {X 0,Y 62.543,Z 381.232,A -85,B 0,C 180,E1 -28324.014,E2 -28324.014} C_VEL
LIN {X 0,Y 62.299,Z 378.155,A -85,B 0,C 180,E1 -28333.62,E2 -28333.62} C_VEL
LIN {X 0,Y 63.625,Z 373.7,A -85,B 0,C 180,E1 -28343.76,E2 -28343.76} C_VEL
LIN {X 0,Y 66.213,Z 368.141,A -85,B 0,C 180,E1 -28353.043,E2 -28353.043} C_VEL
LIN {X 0,Y 70.1,Z 361.133,A -85,B 0,C 180,E1 -28361.568,E2 -28361.568} C_VEL
LIN {X 0,Y 74.551,Z 353.442,A -85,B 0,C 180,E1 -28368.346,E2 -28368.346} C_VEL
LIN {X 0,Y 79.116,Z 345.35,A -85,B 0,C 180,E1 -28373.563,E2 -28373.563} C_VEL
LIN {X 0,Y 84.664,Z 334.625,A -85,B 0,C 180,E1 -28378.511,E2 -28378.511} C_VEL
LIN {X 0,Y 89.385,Z 324.012,A -85,B 0,C 180,E1 -28382.056,E2 -28382.056} C_VEL
LIN {X 0,Y 93.395,Z 313.417,A -85,B 0,C 180,E1 -28384.622,E2 -28384.622} C_VEL
LIN {X 0,Y 97.063,Z 301.082,A -85,B 0,C 180,E1 -28386.787,E2 -28386.787} C_VEL
LIN {X 0,Y 99.845,Z 288.055,A -85,B 0,C 180,E1 -28388.342,E2 -28388.342} C_VEL
LIN {X 0,Y 101.682,Z 275.101,A -85,B 0,C 180,E1 -28389.239,E2 -28389.239} C_VEL
LIN {X 0,Y 104.387,Z 246.053,A -85,B 0,C 180,E1 -28390.669,E2 -28390.669} C_VEL
LIN {X 0,Y 100.588,Z 236.974,A -85,B 0,C 180,E1 -28394.668,E2 -28394.668} C_VEL
LIN {X 0,Y 96.686,Z 229.257,A -85,B 0,C 180,E1 -28399.402,E2 -28399.402} C_VEL
LIN {X 0,Y 94.331,Z 225.285,A -85,B 0,C 180,E1 -28402.733,E2 -28402.733} C_VEL
LIN {X 0,Y 92.383,Z 222.008,A -85,B 0,C 180,E1 -28405.973,E2 -28405.973} C_VEL
LIN {X 0,Y 90.372,Z 218.661,A -85,B 0,C 180,E1 -28409.961,E2 -28409.961} C_VEL
LIN {X 0,Y 88.081,Z 215.367,A -85,B 0,C 180,E1 -28415.872,E2 -28415.872} C_VEL
LIN {X 0,Y 87.642,Z 214.277,A -85,B 0,C 180,E1 -28417.554,E2 -28417.554} C_VEL
LIN {X 0,Y 85.989,Z 212.477,A -85,B 0,C 180,E1 -28430.595,E2 -28430.595} C_VEL
LIN {X 0,Y 87.029,Z 213.218,A -85,B 0,C 180,E1 -28439.28,E2 -28439.28} C_VEL
LIN {X 0,Y 88.081,Z 214.339,A -85,B 0,C 180,E1 -28443.219,E2 -28443.219} C_VEL
LIN {X 0,Y 90.159,Z 218.118,A -85,B 0,C 180,E1 -28448.972,E2 -28448.972} C_VEL
LIN {X 0,Y 90.967,Z 219.454,A -85,B 0,C 180,E1 -28450.719,E2 -28450.719} C_VEL
LIN {X 0,Y 93.656,Z 223.93,A -85,B 0,C 180,E1 -28455.647,E2 -28455.647} C_VEL
LIN {X 0,Y 96.266,Z 228.43,A -85,B 0,C 180,E1 -28459.499,E2 -28459.499} C_VEL
LIN {X 0,Y 100.141,Z 236.132,A -85,B 0,C 180,E1 -28464.314,E2 -28464.314} C_VEL
LIN {X 0,Y 101.865,Z 240.381,A -85,B 0,C 180,E1 -28466.265,E2 -28466.265} C_VEL
LIN {X 0,Y 104.187,Z 249.26,A -85,B 0,C 180,E1 -28469.03,E2 -28469.03} C_VEL
LIN {X 0,Y 100.656,Z 286.101,A -85,B 0,C 180,E1 -28470.961,E2 -28470.961} C_VEL
LIN {X 0,Y 98.118,Z 299.873,A -85,B 0,C 180,E1 -28472.207,E2 -28472.207} C_VEL
LIN {X 0,Y 94.74,Z 312.261,A -85,B 0,C 180,E1 -28473.909,E2 -28473.909} C_VEL
LIN {X 0,Y 90.546,Z 324.187,A -85,B 0,C 180,E1 -28476.36,E2 -28476.36} C_VEL
LIN {X 0,Y 86.151,Z 334.324,A -85,B 0,C 180,E1 -28479.194,E2 -28479.194} C_VEL
LIN {X 0,Y 81.463,Z 343.807,A -85,B 0,C 180,E1 -28482.833,E2 -28482.833} C_VEL
LIN {X 0,Y 77.505,Z 351.303,A -85,B 0,C 180,E1 -28486.72,E2 -28486.72} C_VEL
LIN {X 0,Y 72.544,Z 359.987,A -85,B 0,C 180,E1 -28492.734,E2 -28492.734} C_VEL
LIN {X 0,Y 68.016,Z 368.067,A -85,B 0,C 180,E1 -28500.605,E2 -28500.605} C_VEL
LIN {X 0,Y 65.225,Z 373.503,A -85,B 0,C 180,E1 -28507.843,E2 -28507.843} C_VEL
LIN {X 0,Y 63.305,Z 378.807,A -85,B 0,C 180,E1 -28517.17,E2 -28517.17} C_VEL
LIN {X 0,Y 62.767,Z 382.878,A -85,B 0,C 180,E1 -28526.789,E2 -28526.789} C_VEL
LIN {X 0,Y 62.877,Z 383.966,A -85,B 0,C 180,E1 -28529.999,E2 -28529.999} C_VEL
LIN {X 0,Y 62.857,Z 385.794,A -85,B 0,C 180,E1 -28536.419,E2 -28536.419} C_VEL
LIN {X 0,Y 63.347,Z 387.191,A -85,B 0,C 180,E1 -28542.819,E2 -28542.819} C_VEL
LIN {X 0,Y 66.431,Z 388.751,A -85,B 0,C 180,E1 -28555.034,E2 -28555.034} C_VEL
LIN {X 0,Y 72.265,Z 388.837,A -85,B 0,C 180,E1 -28565.697,E2 -28565.697} C_VEL
LIN {X 0,Y 76.05,Z 388.309,A -85,B 0,C 180,E1 -28570.307,E2 -28570.307} C_VEL
LIN {X 0,Y 84.936,Z 386.072,A -85,B 0,C 180,E1 -28578.133,E2 -28578.133} C_VEL
LIN {X 0,Y 92.432,Z 383.359,A -85,B 0,C 180,E1 -28582.973,E2 -28582.973} C_VEL
LIN {X 0,Y 100.555,Z 379.676,A -85,B 0,C 180,E1 -28587.003,E2 -28587.003} C_VEL
LIN {X 0,Y 109.188,Z 374.921,A -85,B 0,C 180,E1 -28590.335,E2 -28590.335} C_VEL
LIN {X 0,Y 118.188,Z 368.951,A -85,B 0,C 180,E1 -28593.121,E2 -28593.121} C_VEL
LIN {X 0,Y 127.422,Z 361.56,A -85,B 0,C 180,E1 -28595.513,E2 -28595.513} C_VEL
LIN {X 0,Y 136.847,Z 352.423,A -85,B 0,C 180,E1 -28597.581,E2 -28597.581} C_VEL
LIN {X 0,Y 145.725,Z 341.9,A -85,B 0,C 180,E1 -28599.133,E2 -28599.133} C_VEL
LIN {X 0,Y 153.092,Z 331.229,A -85,B 0,C 180,E1 -28600.236,E2 -28600.236} C_VEL
LIN {X 0,Y 159.552,Z 319.468,A -85,B 0,C 180,E1 -28601.101,E2 -28601.101} C_VEL
LIN {X 0,Y 164.89,Z 306.868,A -85,B 0,C 180,E1 -28601.764,E2 -28601.764} C_VEL
LIN {X 0,Y 167.191,Z 300.049,A -85,B 0,C 180,E1 -28602.019,E2 -28602.019} C_VEL
LIN {X 0,Y 167.396,Z 298.867,A -85,B 0,C 180,E1 -28602.358,E2 -28602.358} C_VEL
LIN {X 0,Y 167.22,Z 296.309,A -85,B 0,C 180,E1 -28604.833,E2 -28604.833} C_VEL
LIN {X 0,Y 167.067,Z 294.129,A -85,B 0,C 180,E1 -28608.472,E2 -28608.472} C_VEL
LIN {X 0,Y 167.153,Z 294.122,A -85,B 0,C 180,E1 -28613.359,E2 -28613.359} C_VEL
LIN {X 0,Y 167.463,Z 297.541,A -85,B 0,C 180,E1 -28618.107,E2 -28618.107} C_VEL
LIN {X 0,Y 167.478,Z 298.013,A -85,B 0,C 180,E1 -28618.493,E2 -28618.493} C_VEL
LIN {X 0,Y 162.929,Z 310.758,A -85,B 0,C 180,E1 -28619.2,E2 -28619.2} C_VEL
LIN {X 0,Y 162.58,Z 311.586,A -85,B 0,C 180,E1 -28619.251,E2 -28619.251} C_VEL
LIN {X 0,Y 160.081,Z 316.958,A -85,B 0,C 180,E1 -28619.38,E2 -28619.38} C_VEL
LIN {X 0,Y 155.173,Z 325.528,A -85,B 0,C 180,E1 -28619.044,E2 -28619.044} C_VEL
LIN {X 0,Y 149.65,Z 333.709,A -85,B 0,C 180,E1 -28618.778,E2 -28618.778} C_VEL
LIN {X 0,Y 146.178,Z 338.412,A -85,B 0,C 180,E1 -28619.053,E2 -28619.053} C_VEL
LIN {X 0,Y 138.805,Z 347.368,A -85,B 0,C 180,E1 -28620.345,E2 -28620.345} C_VEL
LIN {X 0,Y 130.099,Z 356.099,A -85,B 0,C 180,E1 -28622.026,E2 -28622.026} C_VEL
LIN {X 0,Y 119.826,Z 364.557,A -85,B 0,C 180,E1 -28624.382,E2 -28624.382} C_VEL
LIN {X 0,Y 110.748,Z 370.641,A -85,B 0,C 180,E1 -28626.905,E2 -28626.905} C_VEL
LIN {X 0,Y 100.082,Z 376.37,A -85,B 0,C 180,E1 -28630.547,E2 -28630.547} C_VEL
LIN {X 0,Y 90.792,Z 380.28,A -85,B 0,C 180,E1 -28634.626,E2 -28634.626} C_VEL
LIN {X 0,Y 81.09,Z 383.291,A -85,B 0,C 180,E1 -28640.281,E2 -28640.281} C_VEL
LIN {X 0,Y 76.662,Z 384.275,A -85,B 0,C 180,E1 -28643.546,E2 -28643.546} C_VEL
LIN {X 0,Y 69.522,Z 385.229,A -85,B 0,C 180,E1 -28650.357,E2 -28650.357} C_VEL
LIN {X 0,Y 63.238,Z 385.194,A -85,B 0,C 180,E1 -28658.928,E2 -28658.928} C_VEL
LIN {X 0,Y 60.017,Z 384.583,A -85,B 0,C 180,E1 -28665.365,E2 -28665.365} C_VEL
LIN {X 0,Y 57.537,Z 383.528,A -85,B 0,C 180,E1 -28672.358,E2 -28672.358} C_VEL
LIN {X 0,Y 55.598,Z 381.46,A -85,B 0,C 180,E1 -28682.224,E2 -28682.224} C_VEL
LIN {X 0,Y 55.287,Z 377.601,A -85,B 0,C 180,E1 -28695.273,E2 -28695.273} C_VEL
LIN {X 0,Y 57.141,Z 372.639,A -85,B 0,C 180,E1 -28707.149,E2 -28707.149} C_VEL
LIN {X 0,Y 60.772,Z 365.965,A -85,B 0,C 180,E1 -28718.313,E2 -28718.313} C_VEL
LIN {X 0,Y 65.547,Z 358.338,A -85,B 0,C 180,E1 -28727.15,E2 -28727.15} C_VEL
LIN {X 0,Y 70.429,Z 350.557,A -85,B 0,C 180,E1 -28733.526,E2 -28733.526} C_VEL
LIN {X 0,Y 75.99,Z 341.105,A -85,B 0,C 180,E1 -28739.05,E2 -28739.05} C_VEL
LIN {X 0,Y 81.455,Z 330.543,A -85,B 0,C 180,E1 -28743.371,E2 -28743.371} C_VEL
LIN {X 0,Y 86.62,Z 318.808,A -85,B 0,C 180,E1 -28746.755,E2 -28746.755} C_VEL
LIN {X 0,Y 90.417,Z 308.099,A -85,B 0,C 180,E1 -28748.991,E2 -28748.991} C_VEL
LIN {X 0,Y 93.935,Z 295.346,A -85,B 0,C 180,E1 -28750.81,E2 -28750.81} C_VEL
LIN {X 0,Y 96.491,Z 281.509,A -85,B 0,C 180,E1 -28752.108,E2 -28752.108} C_VEL
LIN {X 0,Y 99.929,Z 248.923,A -85,B 0,C 180,E1 -28753.677,E2 -28753.677} C_VEL
LIN {X 0,Y 97.294,Z 241.954,A -85,B 0,C 180,E1 -28756.919,E2 -28756.919} C_VEL
LIN {X 0,Y 93.986,Z 234.815,A -85,B 0,C 180,E1 -28761.501,E2 -28761.501} C_VEL
LIN {X 0,Y 90.771,Z 228.789,A -85,B 0,C 180,E1 -28766.996,E2 -28766.996} C_VEL
LIN {X 0,Y 88.537,Z 225,A -85,B 0,C 180,E1 -28771.832,E2 -28771.832} C_VEL
LIN {X 0,Y 86.646,Z 221.813,A -85,B 0,C 180,E1 -28777.581,E2 -28777.581} C_VEL
LIN {X 0,Y 86.466,Z 221.213,A -85,B 0,C 180,E1 -28778.428,E2 -28778.428} C_VEL
LIN {X 0,Y 85.082,Z 219.532,A -85,B 0,C 180,E1 -28790.493,E2 -28790.493} C_VEL
LIN {X 0,Y 85.957,Z 220.12,A -85,B 0,C 180,E1 -28798.538,E2 -28798.538} C_VEL
LIN {X 0,Y 86.762,Z 221.189,A -85,B 0,C 180,E1 -28801.997,E2 -28801.997} C_VEL
LIN {X 0,Y 89.1,Z 225.699,A -85,B 0,C 180,E1 -28808.912,E2 -28808.912} C_VEL
LIN {X 0,Y 91.601,Z 230.282,A -85,B 0,C 180,E1 -28814.052,E2 -28814.052} C_VEL
LIN {X 0,Y 94.085,Z 235.003,A -85,B 0,C 180,E1 -28818.125,E2 -28818.125} C_VEL
LIN {X 0,Y 97.574,Z 242.689,A -85,B 0,C 180,E1 -28822.919,E2 -28822.919} C_VEL
LIN {X 0,Y 99.128,Z 248.209,A -85,B 0,C 180,E1 -28825.038,E2 -28825.038} C_VEL
LIN {X 0,Y 99.802,Z 251.226,A -85,B 0,C 180,E1 -28825.982,E2 -28825.982} C_VEL
LIN {X 0,Y 96.247,Z 285.941,A -85,B 0,C 180,E1 -28827.744,E2 -28827.744} C_VEL
LIN {X 0,Y 93.605,Z 299.55,A -85,B 0,C 180,E1 -28828.932,E2 -28828.932} C_VEL
LIN {X 0,Y 90.251,Z 311.425,A -85,B 0,C 180,E1 -28830.517,E2 -28830.517} C_VEL
LIN {X 0,Y 85.829,Z 323.503,A -85,B 0,C 180,E1 -28832.931,E2 -28832.931} C_VEL
LIN {X 0,Y 81.169,Z 333.711,A -85,B 0,C 180,E1 -28835.733,E2 -28835.733} C_VEL
LIN {X 0,Y 75.593,Z 344.344,A -85,B 0,C 180,E1 -28839.911,E2 -28839.911} C_VEL
LIN {X 0,Y 71.264,Z 351.767,A -85,B 0,C 180,E1 -28843.953,E2 -28843.953} C_VEL
LIN {X 0,Y 66.035,Z 360.277,A -85,B 0,C 180,E1 -28850.313,E2 -28850.313} C_VEL
LIN {X 0,Y 61.171,Z 368.241,A -85,B 0,C 180,E1 -28858.866,E2 -28858.866} C_VEL
LIN {X 0,Y 57.72,Z 374.558,A -85,B 0,C 180,E1 -28868.574,E2 -28868.574} C_VEL
LIN {X 0,Y 55.978,Z 379.556,A -85,B 0,C 180,E1 -28879.144,E2 -28879.144} C_VEL
LIN {X 0,Y 55.797,Z 383.365,A -85,B 0,C 180,E1 -28889.999,E2 -28889.999} C_VEL
LIN {X 0,Y 55.827,Z 385.248,A -85,B 0,C 180,E1 -28897.231,E2 -28897.231} C_VEL
LIN {X 0,Y 56.455,Z 386.71,A -85,B 0,C 180,E1 -28904.416,E2 -28904.416} C_VEL
LIN {X 0,Y 57.849,Z 387.767,A -85,B 0,C 180,E1 -28911.373,E2 -28911.373} C_VEL
LIN {X 0,Y 62.954,Z 388.688,A -85,B 0,C 180,E1 -28923.929,E2 -28923.929} C_VEL
LIN {X 0,Y 70.765,Z 388.149,A -85,B 0,C 180,E1 -28934.042,E2 -28934.042} C_VEL
LIN {X 0,Y 75.413,Z 387.3,A -85,B 0,C 180,E1 -28938.205,E2 -28938.205} C_VEL
LIN {X 0,Y 85.605,Z 384.405,A -85,B 0,C 180,E1 -28945.183,E2 -28945.183} C_VEL
LIN {X 0,Y 93.957,Z 381.16,A -85,B 0,C 180,E1 -28949.339,E2 -28949.339} C_VEL
LIN {X 0,Y 102.819,Z 376.892,A -85,B 0,C 180,E1 -28952.696,E2 -28952.696} C_VEL
LIN {X 0,Y 113.601,Z 370.479,A -85,B 0,C 180,E1 -28955.855,E2 -28955.855} C_VEL
LIN {X 0,Y 123.056,Z 363.54,A -85,B 0,C 180,E1 -28958.136,E2 -28958.136} C_VEL
LIN {X 0,Y 132.699,Z 354.905,A -85,B 0,C 180,E1 -28960.063,E2 -28960.063} C_VEL
LIN {X 0,Y 140.886,Z 346.092,A -85,B 0,C 180,E1 -28961.406,E2 -28961.406} C_VEL
LIN {X 0,Y 149.187,Z 335.261,A -85,B 0,C 180,E1 -28962.544,E2 -28962.544} C_VEL
LIN {X 0,Y 155.826,Z 324.452,A -85,B 0,C 180,E1 -28963.35,E2 -28963.35} C_VEL
LIN {X 0,Y 161.6,Z 312.579,A -85,B 0,C 180,E1 -28963.992,E2 -28963.992} C_VEL
LIN {X 0,Y 164.684,Z 304.716,A -85,B 0,C 180,E1 -28964.292,E2 -28964.292} C_VEL
LIN {X 0,Y 164.975,Z 303.611,A -85,B 0,C 180,E1 -28964.557,E2 -28964.557} C_VEL
LIN {X 0,Y 165.005,Z 302.95,A -85,B 0,C 180,E1 -28965.192,E2 -28965.192} C_VEL
LIN {X 0,Y 165.001,Z 300.957,A -85,B 0,C 180,E1 -28968.422,E2 -28968.422} C_VEL
LIN {X 0,Y 165.014,Z 300.795,A -85,B 0,C 180,E1 -28972.658,E2 -28972.658} C_VEL
LIN {X 0,Y 164.953,Z 302.845,A -85,B 0,C 180,E1 -28975.943,E2 -28975.943} C_VEL
LIN {X 0,Y 164.607,Z 304.135,A -85,B 0,C 180,E1 -28976.339,E2 -28976.339} C_VEL
LIN {X 0,Y 159.392,Z 316.619,A -85,B 0,C 180,E1 -28977.073,E2 -28977.073} C_VEL
LIN {X 0,Y 152.95,Z 328.486,A -85,B 0,C 180,E1 -28978.021,E2 -28978.021} C_VEL
LIN {X 0,Y 146.178,Z 338.412,A -85,B 0,C 180,E1 -28979.053,E2 -28979.053} C_VEL
LIN {X 0,Y 142.477,Z 342.998,A -85,B 0,C 180,E1 -28979.375,E2 -28979.375} C_VEL
LIN {X 0,Y 132.755,Z 352.928,A -85,B 0,C 180,E1 -28979.224,E2 -28979.224} C_VEL
LIN {X 0,Y 126.83,Z 358.116,A -85,B 0,C 180,E1 -28979.418,E2 -28979.418} C_VEL
LIN {X 0,Y 123.895,Z 360.493,A -85,B 0,C 180,E1 -28979.844,E2 -28979.844} C_VEL
LIN {X 0,Y 114.267,Z 367.518,A -85,B 0,C 180,E1 -28981.9,E2 -28981.9} C_VEL
LIN {X 0,Y 105.694,Z 372.666,A -85,B 0,C 180,E1 -28984.129,E2 -28984.129} C_VEL
LIN {X 0,Y 95.654,Z 377.577,A -85,B 0,C 180,E1 -28987.306,E2 -28987.306} C_VEL
LIN {X 0,Y 85.984,Z 381.235,A -85,B 0,C 180,E1 -28991.239,E2 -28991.239} C_VEL
LIN {X 0,Y 77.481,Z 383.591,A -85,B 0,C 180,E1 -28995.787,E2 -28995.787} C_VEL
LIN {X 0,Y 68.38,Z 385.196,A -85,B 0,C 180,E1 -29002.332,E2 -29002.332} C_VEL
LIN {X 0,Y 63.282,Z 385.567,A -85,B 0,C 180,E1 -29007.32,E2 -29007.32} C_VEL
LIN {X 0,Y 58.718,Z 385.507,A -85,B 0,C 180,E1 -29013.089,E2 -29013.089} C_VEL
LIN {X 0,Y 54.652,Z 384.987,A -85,B 0,C 180,E1 -29020.009,E2 -29020.009} C_VEL
LIN {X 0,Y 51.689,Z 384.038,A -85,B 0,C 180,E1 -29027.171,E2 -29027.171} C_VEL
LIN {X 0,Y 48.724,Z 381.688,A -85,B 0,C 180,E1 -29039.925,E2 -29039.925} C_VEL
LIN {X 0,Y 48.08,Z 378.373,A -85,B 0,C 180,E1 -29053.003,E2 -29053.003} C_VEL
LIN {X 0,Y 49.914,Z 373.233,A -85,B 0,C 180,E1 -29067.484,E2 -29067.484} C_VEL
LIN {X 0,Y 53.574,Z 367.097,A -85,B 0,C 180,E1 -29079.439,E2 -29079.439} C_VEL
LIN {X 0,Y 58.589,Z 359.668,A -85,B 0,C 180,E1 -29089.262,E2 -29089.262} C_VEL
LIN {X 0,Y 64.963,Z 350.414,A -85,B 0,C 180,E1 -29097.375,E2 -29097.375} C_VEL
LIN {X 0,Y 71.004,Z 340.837,A -85,B 0,C 180,E1 -29102.984,E2 -29102.984} C_VEL
LIN {X 0,Y 76.875,Z 330.157,A -85,B 0,C 180,E1 -29107.278,E2 -29107.278} C_VEL
LIN {X 0,Y 82.351,Z 318.279,A -85,B 0,C 180,E1 -29110.598,E2 -29110.598} C_VEL
LIN {X 0,Y 86.777,Z 305.976,A -85,B 0,C 180,E1 -29112.985,E2 -29112.985} C_VEL
LIN {X 0,Y 90.342,Z 292.886,A -85,B 0,C 180,E1 -29114.667,E2 -29114.667} C_VEL
LIN {X 0,Y 92.634,Z 280.018,A -85,B 0,C 180,E1 -29115.745,E2 -29115.745} C_VEL
LIN {X 0,Y 95.688,Z 251.088,A -85,B 0,C 180,E1 -29117.139,E2 -29117.139} C_VEL
LIN {X 0,Y 93.165,Z 244.407,A -85,B 0,C 180,E1 -29120.842,E2 -29120.842} C_VEL
LIN {X 0,Y 90.682,Z 238.882,A -85,B 0,C 180,E1 -29125.029,E2 -29125.029} C_VEL
LIN {X 0,Y 88.339,Z 234.28,A -85,B 0,C 180,E1 -29129.802,E2 -29129.802} C_VEL
LIN {X 0,Y 86.916,Z 231.528,A -85,B 0,C 180,E1 -29133.451,E2 -29133.451} C_VEL
LIN {X 0,Y 85.176,Z 228.062,A -85,B 0,C 180,E1 -29139.894,E2 -29139.894} C_VEL
LIN {X 0,Y 84.177,Z 226.592,A -85,B 0,C 180,E1 -29150.39,E2 -29150.39} C_VEL
LIN {X 0,Y 85.031,Z 227.24,A -85,B 0,C 180,E1 -29158.523,E2 -29158.523} C_VEL
LIN {X 0,Y 85.498,Z 228.001,A -85,B 0,C 180,E1 -29160.761,E2 -29160.761} C_VEL
LIN {X 0,Y 87.485,Z 232.311,A -85,B 0,C 180,E1 -29167.482,E2 -29167.482} C_VEL
LIN {X 0,Y 89.586,Z 236.531,A -85,B 0,C 180,E1 -29172.31,E2 -29172.31} C_VEL
LIN {X 0,Y 91.609,Z 240.82,A -85,B 0,C 180,E1 -29176.096,E2 -29176.096} C_VEL
LIN {X 0,Y 94.468,Z 247.819,A -85,B 0,C 180,E1 -29180.616,E2 -29180.616} C_VEL
LIN {X 0,Y 95.68,Z 253.078,A -85,B 0,C 180,E1 -29182.615,E2 -29182.615} C_VEL
LIN {X 0,Y 92.092,Z 286.118,A -85,B 0,C 180,E1 -29184.249,E2 -29184.249} C_VEL
LIN {X 0,Y 89.268,Z 299.817,A -85,B 0,C 180,E1 -29185.402,E2 -29185.402} C_VEL
LIN {X 0,Y 85.736,Z 311.625,A -85,B 0,C 180,E1 -29186.941,E2 -29186.941} C_VEL
LIN {X 0,Y 81.455,Z 322.792,A -85,B 0,C 180,E1 -29189.119,E2 -29189.119} C_VEL
LIN {X 0,Y 75.856,Z 334.391,A -85,B 0,C 180,E1 -29192.281,E2 -29192.281} C_VEL
LIN {X 0,Y 69.956,Z 344.867,A -85,B 0,C 180,E1 -29196.513,E2 -29196.513} C_VEL
LIN {X 0,Y 65.049,Z 352.504,A -85,B 0,C 180,E1 -29200.86,E2 -29200.86} C_VEL
LIN {X 0,Y 59.68,Z 360.557,A -85,B 0,C 180,E1 -29207.378,E2 -29207.378} C_VEL
LIN {X 0,Y 54.379,Z 368.385,A -85,B 0,C 180,E1 -29216.681,E2 -29216.681} C_VEL
LIN {X 0,Y 50.218,Z 375.543,A -85,B 0,C 180,E1 -29229.519,E2 -29229.519} C_VEL
LIN {X 0,Y 48.7,Z 380.264,A -85,B 0,C 180,E1 -29241.701,E2 -29241.701} C_VEL
LIN {X 0,Y 48.715,Z 382.763,A -85,B 0,C 180,E1 -29249.999,E2 -29249.999} C_VEL
LIN {X 0,Y 48.791,Z 384.7,A -85,B 0,C 180,E1 -29258.28,E2 -29258.28} C_VEL
LIN {X 0,Y 51.292,Z 387.34,A -85,B 0,C 180,E1 -29274.27,E2 -29274.27} C_VEL
LIN {X 0,Y 53.85,Z 388.072,A -85,B 0,C 180,E1 -29281.468,E2 -29281.468} C_VEL
LIN {X 0,Y 61.274,Z 388.368,A -85,B 0,C 180,E1 -29293.485,E2 -29293.485} C_VEL
LIN {X 0,Y 70.863,Z 387.197,A -85,B 0,C 180,E1 -29302.505,E2 -29302.505} C_VEL
LIN {X 0,Y 78.038,Z 385.508,A -85,B 0,C 180,E1 -29307.289,E2 -29307.289} C_VEL
LIN {X 0,Y 90.542,Z 381.31,A -85,B 0,C 180,E1 -29313.206,E2 -29313.206} C_VEL
LIN {X 0,Y 99.769,Z 377.175,A -85,B 0,C 180,E1 -29316.312,E2 -29316.312} C_VEL
LIN {X 0,Y 110.898,Z 370.906,A -85,B 0,C 180,E1 -29319.189,E2 -29319.189} C_VEL
LIN {X 0,Y 120.609,Z 364.13,A -85,B 0,C 180,E1 -29321.245,E2 -29321.245} C_VEL
LIN {X 0,Y 130.465,Z 355.75,A -85,B 0,C 180,E1 -29322.974,E2 -29322.974} C_VEL
LIN {X 0,Y 138.803,Z 347.155,A -85,B 0,C 180,E1 -29324.159,E2 -29324.159} C_VEL
LIN {X 0,Y 147.221,Z 336.606,A -85,B 0,C 180,E1 -29325.169,E2 -29325.169} C_VEL
LIN {X 0,Y 153.919,Z 326.304,A -85,B 0,C 180,E1 -29325.854,E2 -29325.854} C_VEL
LIN {X 0,Y 159.827,Z 314.945,A -85,B 0,C 180,E1 -29326.415,E2 -29326.415} C_VEL
LIN {X 0,Y 161.91,Z 310.153,A -85,B 0,C 180,E1 -29326.593,E2 -29326.593} C_VEL
LIN {X 0,Y 162.446,Z 308.335,A -85,B 0,C 180,E1 -29327.506,E2 -29327.506} C_VEL
LIN {X 0,Y 162.49,Z 307.468,A -85,B 0,C 180,E1 -29330.036,E2 -29330.036} C_VEL
LIN {X 0,Y 162.535,Z 307.545,A -85,B 0,C 180,E1 -29332.545,E2 -29332.545} C_VEL
LIN {X 0,Y 162.408,Z 308.281,A -85,B 0,C 180,E1 -29333.788,E2 -29333.788} C_VEL
LIN {X 0,Y 162.15,Z 309.064,A -85,B 0,C 180,E1 -29334.09,E2 -29334.09} C_VEL
LIN {X 0,Y 156.213,Z 321.618,A -85,B 0,C 180,E1 -29334.836,E2 -29334.836} C_VEL
LIN {X 0,Y 148.871,Z 333.642,A -85,B 0,C 180,E1 -29335.776,E2 -29335.776} C_VEL
LIN {X 0,Y 140.763,Z 344.133,A -85,B 0,C 180,E1 -29336.922,E2 -29336.922} C_VEL
LIN {X 0,Y 131.828,Z 353.55,A -85,B 0,C 180,E1 -29338.369,E2 -29338.369} C_VEL
LIN {X 0,Y 123.895,Z 360.493,A -85,B 0,C 180,E1 -29339.844,E2 -29339.844} C_VEL
LIN {X 0,Y 119.297,Z 363.978,A -85,B 0,C 180,E1 -29340.46,E2 -29340.46} C_VEL
LIN {X 0,Y 110.96,Z 369.323,A -85,B 0,C 180,E1 -29340.754,E2 -29340.754} C_VEL
LIN {X 0,Y 102.255,Z 373.976,A -85,B 0,C 180,E1 -29341.168,E2 -29341.168} C_VEL
LIN {X 0,Y 97.115,Z 376.362,A -85,B 0,C 180,E1 -29342.104,E2 -29342.104} C_VEL
LIN {X 0,Y 89.268,Z 379.576,A -85,B 0,C 180,E1 -29344.513,E2 -29344.513} C_VEL
LIN {X 0,Y 78.256,Z 383.004,A -85,B 0,C 180,E1 -29348.933,E2 -29348.933} C_VEL
LIN {X 0,Y 71.906,Z 384.383,A -85,B 0,C 180,E1 -29352.212,E2 -29352.212} C_VEL
LIN {X 0,Y 65.836,Z 385.324,A -85,B 0,C 180,E1 -29356.108,E2 -29356.108} C_VEL
LIN {X 0,Y 60.136,Z 385.815,A -85,B 0,C 180,E1 -29360.782,E2 -29360.782} C_VEL
LIN {X 0,Y 54.887,Z 385.821,A -85,B 0,C 180,E1 -29366.324,E2 -29366.324} C_VEL
LIN {X 0,Y 49.124,Z 385.23,A -85,B 0,C 180,E1 -29374.903,E2 -29374.903} C_VEL
LIN {X 0,Y 43.412,Z 383.195,A -85,B 0,C 180,E1 -29389.644,E2 -29389.644} C_VEL
LIN {X 0,Y 41.102,Z 380.325,A -85,B 0,C 180,E1 -29404.694,E2 -29404.694} C_VEL
LIN {X 0,Y 41.48,Z 376.357,A -85,B 0,C 180,E1 -29420.247,E2 -29420.247} C_VEL
LIN {X 0,Y 44.259,Z 371.211,A -85,B 0,C 180,E1 -29434.555,E2 -29434.555} C_VEL
LIN {X 0,Y 48.955,Z 364.759,A -85,B 0,C 180,E1 -29446.687,E2 -29446.687} C_VEL
LIN {X 0,Y 54.841,Z 357.02,A -85,B 0,C 180,E1 -29456.235,E2 -29456.235} C_VEL
LIN {X 0,Y 61.109,Z 348.459,A -85,B 0,C 180,E1 -29463.114,E2 -29463.114} C_VEL
LIN {X 0,Y 67.783,Z 338.368,A -85,B 0,C 180,E1 -29468.471,E2 -29468.471} C_VEL
LIN {X 0,Y 73.383,Z 328.462,A -85,B 0,C 180,E1 -29472.1,E2 -29472.1} C_VEL
LIN {X 0,Y 78.499,Z 317.686,A -85,B 0,C 180,E1 -29474.835,E2 -29474.835} C_VEL
LIN {X 0,Y 82.961,Z 305.711,A -85,B 0,C 180,E1 -29477.027,E2 -29477.027} C_VEL
LIN {X 0,Y 86.544,Z 293.05,A -85,B 0,C 180,E1 -29478.553,E2 -29478.553} C_VEL
LIN {X 0,Y 88.967,Z 279.99,A -85,B 0,C 180,E1 -29479.572,E2 -29479.572} C_VEL
LIN {X 0,Y 91.87,Z 253.871,A -85,B 0,C 180,E1 -29480.752,E2 -29480.752} C_VEL
LIN {X 0,Y 89.53,Z 247.278,A -85,B 0,C 180,E1 -29484.998,E2 -29484.998} C_VEL
LIN {X 0,Y 87.498,Z 242.658,A -85,B 0,C 180,E1 -29489.263,E2 -29489.263} C_VEL
LIN {X 0,Y 85.576,Z 238.318,A -85,B 0,C 180,E1 -29494.501,E2 -29494.501} C_VEL
LIN {X 0,Y 83.983,Z 234.919,A -85,B 0,C 180,E1 -29501.215,E2 -29501.215} C_VEL
LIN {X 0,Y 83.274,Z 233.634,A -85,B 0,C 180,E1 -29510.285,E2 -29510.285} C_VEL
LIN {X 0,Y 83.982,Z 234.181,A -85,B 0,C 180,E1 -29517.808,E2 -29517.808} C_VEL
LIN {X 0,Y 84.338,Z 235.003,A -85,B 0,C 180,E1 -29519.835,E2 -29519.835} C_VEL
LIN {X 0,Y 85.8,Z 238.609,A -85,B 0,C 180,E1 -29525.606,E2 -29525.606} C_VEL
LIN {X 0,Y 87.759,Z 243.012,A -85,B 0,C 180,E1 -29530.736,E2 -29530.736} C_VEL
LIN {X 0,Y 89.837,Z 248.12,A -85,B 0,C 180,E1 -29535.094,E2 -29535.094} C_VEL
LIN {X 0,Y 91.465,Z 252.886,A -85,B 0,C 180,E1 -29538.078,E2 -29538.078} C_VEL
LIN {X 0,Y 91.88,Z 255.035,A -85,B 0,C 180,E1 -29538.934,E2 -29538.934} C_VEL
LIN {X 0,Y 88.357,Z 286.004,A -85,B 0,C 180,E1 -29540.416,E2 -29540.416} C_VEL
LIN {X 0,Y 85.48,Z 299.435,A -85,B 0,C 180,E1 -29541.478,E2 -29541.478} C_VEL
LIN {X 0,Y 81.594,Z 311.805,A -85,B 0,C 180,E1 -29542.989,E2 -29542.989} C_VEL
LIN {X 0,Y 76.723,Z 323.666,A -85,B 0,C 180,E1 -29545.231,E2 -29545.231} C_VEL
LIN {X 0,Y 71.564,Z 333.757,A -85,B 0,C 180,E1 -29547.886,E2 -29547.886} C_VEL
LIN {X 0,Y 65.207,Z 344.389,A -85,B 0,C 180,E1 -29552.043,E2 -29552.043} C_VEL
LIN {X 0,Y 60.646,Z 351.097,A -85,B 0,C 180,E1 -29555.785,E2 -29555.785} C_VEL
LIN {X 0,Y 54.621,Z 359.328,A -85,B 0,C 180,E1 -29562.28,E2 -29562.28} C_VEL
LIN {X 0,Y 48.587,Z 367.391,A -85,B 0,C 180,E1 -29572.064,E2 -29572.064} C_VEL
LIN {X 0,Y 44.715,Z 372.805,A -85,B 0,C 180,E1 -29581.865,E2 -29581.865} C_VEL
LIN {X 0,Y 42.085,Z 378.089,A -85,B 0,C 180,E1 -29595.492,E2 -29595.492} C_VEL
LIN {X 0,Y 41.617,Z 382.136,A -85,B 0,C 180,E1 -29609.998,E2 -29609.998} C_VEL
LIN {X 0,Y 41.791,Z 384.153,A -85,B 0,C 180,E1 -29619.68,E2 -29619.68} C_VEL
LIN {X 0,Y 44.909,Z 386.898,A -85,B 0,C 180,E1 -29637.999,E2 -29637.999} C_VEL
LIN {X 0,Y 51.763,Z 388.115,A -85,B 0,C 180,E1 -29652.753,E2 -29652.753} C_VEL
LIN {X 0,Y 61.334,Z 387.784,A -85,B 0,C 180,E1 -29663.33,E2 -29663.33} C_VEL
LIN {X 0,Y 72.435,Z 385.982,A -85,B 0,C 180,E1 -29670.834,E2 -29670.834} C_VEL
LIN {X 0,Y 78.351,Z 384.48,A -85,B 0,C 180,E1 -29673.764,E2 -29673.764} C_VEL
LIN {X 0,Y 87.576,Z 381.472,A -85,B 0,C 180,E1 -29677.349,E2 -29677.349} C_VEL
LIN {X 0,Y 97.142,Z 377.455,A -85,B 0,C 180,E1 -29680.138,E2 -29680.138} C_VEL
LIN {X 0,Y 108.588,Z 371.333,A -85,B 0,C 180,E1 -29682.676,E2 -29682.676} C_VEL
LIN {X 0,Y 118.531,Z 364.708,A -85,B 0,C 180,E1 -29684.472,E2 -29684.472} C_VEL
LIN {X 0,Y 128.578,Z 356.534,A -85,B 0,C 180,E1 -29685.977,E2 -29685.977} C_VEL
LIN {X 0,Y 137.05,Z 348.19,A -85,B 0,C 180,E1 -29686.99,E2 -29686.99} C_VEL
LIN {X 0,Y 145.581,Z 337.934,A -85,B 0,C 180,E1 -29687.844,E2 -29687.844} C_VEL
LIN {X 0,Y 152.949,Z 326.994,A -85,B 0,C 180,E1 -29688.461,E2 -29688.461} C_VEL
LIN {X 0,Y 159.049,Z 315.641,A -85,B 0,C 180,E1 -29688.94,E2 -29688.94} C_VEL
LIN {X 0,Y 159.686,Z 314.092,A -85,B 0,C 180,E1 -29689.859,E2 -29689.859} C_VEL
LIN {X 0,Y 159.684,Z 314.031,A -85,B 0,C 180,E1 -29691.265,E2 -29691.265} C_VEL
LIN {X 0,Y 159.468,Z 314.566,A -85,B 0,C 180,E1 -29691.828,E2 -29691.828} C_VEL
LIN {X 0,Y 153.264,Z 326.214,A -85,B 0,C 180,E1 -29692.499,E2 -29692.499} C_VEL
LIN {X 0,Y 145.95,Z 337.096,A -85,B 0,C 180,E1 -29693.297,E2 -29693.297} C_VEL
LIN {X 0,Y 137.828,Z 346.908,A -85,B 0,C 180,E1 -29694.319,E2 -29694.319} C_VEL
LIN {X 0,Y 128.638,Z 355.922,A -85,B 0,C 180,E1 -29695.611,E2 -29695.611} C_VEL
LIN {X 0,Y 117.838,Z 364.501,A -85,B 0,C 180,E1 -29697.418,E2 -29697.418} C_VEL
LIN {X 0,Y 108.944,Z 370.25,A -85,B 0,C 180,E1 -29699.191,E2 -29699.191} C_VEL
LIN {X 0,Y 98.437,Z 375.782,A -85,B 0,C 180,E1 -29701.745,E2 -29701.745} C_VEL
LIN {X 0,Y 97.115,Z 376.362,A -85,B 0,C 180,E1 -29702.104,E2 -29702.104} C_VEL
LIN {X 0,Y 91.887,Z 378.541,A -85,B 0,C 180,E1 -29703.189,E2 -29703.189} C_VEL
LIN {X 0,Y 82.578,Z 381.652,A -85,B 0,C 180,E1 -29704.21,E2 -29704.21} C_VEL
LIN {X 0,Y 73.146,Z 383.963,A -85,B 0,C 180,E1 -29705.588,E2 -29705.588} C_VEL
LIN {X 0,Y 67.817,Z 384.878,A -85,B 0,C 180,E1 -29707.477,E2 -29707.477} C_VEL
LIN {X 0,Y 57.001,Z 386.076,A -85,B 0,C 180,E1 -29714.272,E2 -29714.272} C_VEL
LIN {X 0,Y 46.512,Z 385.777,A -85,B 0,C 180,E1 -29724.963,E2 -29724.963} C_VEL
LIN {X 0,Y 41.756,Z 384.999,A -85,B 0,C 180,E1 -29732.698,E2 -29732.698} C_VEL
LIN {X 0,Y 37.903,Z 383.763,A -85,B 0,C 180,E1 -29742.128,E2 -29742.128} C_VEL
LIN {X 0,Y 34.412,Z 381.027,A -85,B 0,C 180,E1 -29759.3,E2 -29759.3} C_VEL
LIN {X 0,Y 34.123,Z 377.2,A -85,B 0,C 180,E1 -29778.116,E2 -29778.116} C_VEL
LIN {X 0,Y 36.913,Z 372.196,A -85,B 0,C 180,E1 -29795.465,E2 -29795.465} C_VEL
LIN {X 0,Y 41.953,Z 365.91,A -85,B 0,C 180,E1 -29809.577,E2 -29809.577} C_VEL
LIN {X 0,Y 48.32,Z 358.536,A -85,B 0,C 180,E1 -29819.855,E2 -29819.855} C_VEL
LIN {X 0,Y 55.167,Z 350.109,A -85,B 0,C 180,E1 -29827.24,E2 -29827.24} C_VEL
LIN {X 0,Y 62.254,Z 340.299,A -85,B 0,C 180,E1 -29832.639,E2 -29832.639} C_VEL
LIN {X 0,Y 68.959,Z 329.399,A -85,B 0,C 180,E1 -29836.566,E2 -29836.566} C_VEL
LIN {X 0,Y 74.875,Z 317.61,A -85,B 0,C 180,E1 -29839.393,E2 -29839.393} C_VEL
LIN {X 0,Y 79.828,Z 304.784,A -85,B 0,C 180,E1 -29841.516,E2 -29841.516} C_VEL
LIN {X 0,Y 83.534,Z 291.757,A -85,B 0,C 180,E1 -29842.901,E2 -29842.901} C_VEL
LIN {X 0,Y 86.017,Z 278.017,A -85,B 0,C 180,E1 -29843.761,E2 -29843.761} C_VEL
LIN {X 0,Y 88.416,Z 257.18,A -85,B 0,C 180,E1 -29844.602,E2 -29844.602} C_VEL
LIN {X 0,Y 88.026,Z 255.396,A -85,B 0,C 180,E1 -29845.544,E2 -29845.544} C_VEL
LIN {X 0,Y 86.207,Z 250.225,A -85,B 0,C 180,E1 -29849.739,E2 -29849.739} C_VEL
LIN {X 0,Y 84.504,Z 245.983,A -85,B 0,C 180,E1 -29854.646,E2 -29854.646} C_VEL
LIN {X 0,Y 83.786,Z 244.29,A -85,B 0,C 180,E1 -29857.325,E2 -29857.325} C_VEL
LIN {X 0,Y 82.97,Z 241.916,A -85,B 0,C 180,E1 -29861.752,E2 -29861.752} C_VEL
LIN {X 0,Y 82.371,Z 240.686,A -85,B 0,C 180,E1 -29870.178,E2 -29870.178} C_VEL
LIN {X 0,Y 83.038,Z 241.249,A -85,B 0,C 180,E1 -29877.65,E2 -29877.65} C_VEL
LIN {X 0,Y 84.286,Z 245.123,A -85,B 0,C 180,E1 -29883.939,E2 -29883.939} C_VEL
LIN {X 0,Y 86.147,Z 249.886,A -85,B 0,C 180,E1 -29889.522,E2 -29889.522} C_VEL
LIN {X 0,Y 88.199,Z 256.087,A -85,B 0,C 180,E1 -29894.348,E2 -29894.348} C_VEL
LIN {X 0,Y 88.484,Z 257.103,A -85,B 0,C 180,E1 -29894.968,E2 -29894.968} C_VEL
LIN {X 0,Y 85.07,Z 285.792,A -85,B 0,C 180,E1 -29896.261,E2 -29896.261} C_VEL
LIN {X 0,Y 82.097,Z 299.176,A -85,B 0,C 180,E1 -29897.223,E2 -29897.223} C_VEL
LIN {X 0,Y 78.279,Z 310.952,A -85,B 0,C 180,E1 -29898.498,E2 -29898.498} C_VEL
LIN {X 0,Y 73.177,Z 322.952,A -85,B 0,C 180,E1 -29900.539,E2 -29900.539} C_VEL
LIN {X 0,Y 67.745,Z 333.124,A -85,B 0,C 180,E1 -29902.967,E2 -29902.967} C_VEL
LIN {X 0,Y 60.893,Z 343.945,A -85,B 0,C 180,E1 -29906.924,E2 -29906.924} C_VEL
LIN {X 0,Y 55.362,Z 351.48,A -85,B 0,C 180,E1 -29911.028,E2 -29911.028} C_VEL
LIN {X 0,Y 48.834,Z 359.608,A -85,B 0,C 180,E1 -29917.668,E2 -29917.668} C_VEL
LIN {X 0,Y 43.186,Z 366.337,A -85,B 0,C 180,E1 -29926.237,E2 -29926.237} C_VEL
LIN {X 0,Y 38.571,Z 371.89,A -85,B 0,C 180,E1 -29936.862,E2 -29936.862} C_VEL
LIN {X 0,Y 35.233,Z 377.306,A -85,B 0,C 180,E1 -29952.588,E2 -29952.588} C_VEL
LIN {X 0,Y 34.541,Z 381.478,A -85,B 0,C 180,E1 -29969.998,E2 -29969.998} C_VEL
LIN {X 0,Y 34.838,Z 383.596,A -85,B 0,C 180,E1 -29981.636,E2 -29981.636} C_VEL
LIN {X 0,Y 38.766,Z 386.454,A -85,B 0,C 180,E1 -30002.946,E2 -30002.946} C_VEL
LIN {X 0,Y 46.795,Z 387.792,A -85,B 0,C 180,E1 -30018.669,E2 -30018.669} C_VEL
LIN {X 0,Y 51.89,Z 387.901,A -85,B 0,C 180,E1 -30024.353,E2 -30024.353} C_VEL
LIN {X 0,Y 63.211,Z 386.947,A -85,B 0,C 180,E1 -30032.804,E2 -30032.804} C_VEL
LIN {X 0,Y 75.481,Z 384.506,A -85,B 0,C 180,E1 -30038.604,E2 -30038.604} C_VEL
LIN {X 0,Y 85.093,Z 381.588,A -85,B 0,C 180,E1 -30041.768,E2 -30041.768} C_VEL
LIN {X 0,Y 94.968,Z 377.686,A -85,B 0,C 180,E1 -30044.164,E2 -30044.164} C_VEL
LIN {X 0,Y 105,Z 372.698,A -85,B 0,C 180,E1 -30046.054,E2 -30046.054} C_VEL
LIN {X 0,Y 115.14,Z 366.475,A -85,B 0,C 180,E1 -30047.585,E2 -30047.585} C_VEL
LIN {X 0,Y 125.344,Z 358.76,A -85,B 0,C 180,E1 -30048.876,E2 -30048.876} C_VEL
LIN {X 0,Y 133.923,Z 350.906,A -85,B 0,C 180,E1 -30049.725,E2 -30049.725} C_VEL
LIN {X 0,Y 142.535,Z 341.361,A -85,B 0,C 180,E1 -30050.45,E2 -30050.45} C_VEL
LIN {X 0,Y 142.383,Z 341.519,A -85,B 0,C 180,E1 -30050.821,E2 -30050.821} C_VEL
LIN {X 0,Y 133.127,Z 351.584,A -85,B 0,C 180,E1 -30051.827,E2 -30051.827} C_VEL
LIN {X 0,Y 123.962,Z 359.653,A -85,B 0,C 180,E1 -30052.961,E2 -30052.961} C_VEL
LIN {X 0,Y 112.956,Z 367.515,A -85,B 0,C 180,E1 -30054.56,E2 -30054.56} C_VEL
LIN {X 0,Y 101.3,Z 374.113,A -85,B 0,C 180,E1 -30056.697,E2 -30056.697} C_VEL
LIN {X 0,Y 91.378,Z 378.495,A -85,B 0,C 180,E1 -30058.966,E2 -30058.966} C_VEL
LIN {X 0,Y 84.346,Z 380.963,A -85,B 0,C 180,E1 -30060.928,E2 -30060.928} C_VEL
LIN {X 0,Y 77.436,Z 382.955,A -85,B 0,C 180,E1 -30063.307,E2 -30063.307} C_VEL
LIN {X 0,Y 67.817,Z 384.878,A -85,B 0,C 180,E1 -30067.477,E2 -30067.477} C_VEL
LIN {X 0,Y 62.526,Z 385.643,A -85,B 0,C 180,E1 -30069.709,E2 -30069.709} C_VEL
LIN {X 0,Y 53.103,Z 386.258,A -85,B 0,C 180,E1 -30072.709,E2 -30072.709} C_VEL
LIN {X 0,Y 43.854,Z 386.117,A -85,B 0,C 180,E1 -30076.939,E2 -30076.939} C_VEL
LIN {X 0,Y 39.066,Z 385.586,A -85,B 0,C 180,E1 -30081.673,E2 -30081.673} C_VEL
LIN {X 0,Y 33.25,Z 384.296,A -85,B 0,C 180,E1 -30092.281,E2 -30092.281} C_VEL
LIN {X 0,Y 28.981,Z 382.333,A -85,B 0,C 180,E1 -30106.667,E2 -30106.667} C_VEL
LIN {X 0,Y 26.791,Z 379.34,A -85,B 0,C 180,E1 -30126.831,E2 -30126.831} C_VEL
LIN {X 0,Y 28.243,Z 374.883,A -85,B 0,C 180,E1 -30150.003,E2 -30150.003} C_VEL
LIN {X 0,Y 33.083,Z 369.197,A -85,B 0,C 180,E1 -30168.584,E2 -30168.584} C_VEL
LIN {X 0,Y 39.975,Z 362.129,A -85,B 0,C 180,E1 -30181.834,E2 -30181.834} C_VEL
LIN {X 0,Y 46.688,Z 354.926,A -85,B 0,C 180,E1 -30189.776,E2 -30189.776} C_VEL
LIN {X 0,Y 54.078,Z 346.189,A -85,B 0,C 180,E1 -30195.628,E2 -30195.628} C_VEL
LIN {X 0,Y 61.86,Z 335.356,A -85,B 0,C 180,E1 -30200.077,E2 -30200.077} C_VEL
LIN {X 0,Y 68.202,Z 324.631,A -85,B 0,C 180,E1 -30203.001,E2 -30203.001} C_VEL
LIN {X 0,Y 73.648,Z 313.281,A -85,B 0,C 180,E1 -30205.033,E2 -30205.033} C_VEL
LIN {X 0,Y 78.119,Z 300.997,A -85,B 0,C 180,E1 -30206.599,E2 -30206.599} C_VEL
LIN {X 0,Y 81.582,Z 287.678,A -85,B 0,C 180,E1 -30207.716,E2 -30207.716} C_VEL
LIN {X 0,Y 83.682,Z 274.427,A -85,B 0,C 180,E1 -30208.325,E2 -30208.325} C_VEL
LIN {X 0,Y 85.352,Z 259.781,A -85,B 0,C 180,E1 -30208.922,E2 -30208.922} C_VEL
LIN {X 0,Y 84.112,Z 255.714,A -85,B 0,C 180,E1 -30212.49,E2 -30212.49} C_VEL
LIN {X 0,Y 82.743,Z 251.558,A -85,B 0,C 180,E1 -30217.624,E2 -30217.624} C_VEL
LIN {X 0,Y 81.852,Z 248.785,A -85,B 0,C 180,E1 -30223.058,E2 -30223.058} C_VEL
LIN {X 0,Y 81.465,Z 247.766,A -85,B 0,C 180,E1 -30230.067,E2 -30230.067} C_VEL
LIN {X 0,Y 81.929,Z 248.071,A -85,B 0,C 180,E1 -30236.351,E2 -30236.351} C_VEL
LIN {X 0,Y 82.845,Z 251.664,A -85,B 0,C 180,E1 -30242.225,E2 -30242.225} C_VEL
LIN {X 0,Y 84.181,Z 255.7,A -85,B 0,C 180,E1 -30247.12,E2 -30247.12} C_VEL
LIN {X 0,Y 85.443,Z 260.122,A -85,B 0,C 180,E1 -30250.78,E2 -30250.78} C_VEL
LIN {X 0,Y 82.334,Z 285.17,A -85,B 0,C 180,E1 -30251.784,E2 -30251.784} C_VEL
LIN {X 0,Y 79.217,Z 298.784,A -85,B 0,C 180,E1 -30252.598,E2 -30252.598} C_VEL
LIN {X 0,Y 75.078,Z 311.128,A -85,B 0,C 180,E1 -30253.779,E2 -30253.779} C_VEL
LIN {X 0,Y 69.347,Z 323.806,A -85,B 0,C 180,E1 -30255.675,E2 -30255.675} C_VEL
LIN {X 0,Y 62.907,Z 335.105,A -85,B 0,C 180,E1 -30258.26,E2 -30258.26} C_VEL
LIN {X 0,Y 56.616,Z 344.237,A -85,B 0,C 180,E1 -30261.412,E2 -30261.412} C_VEL
LIN {X 0,Y 50.529,Z 351.871,A -85,B 0,C 180,E1 -30265.344,E2 -30265.344} C_VEL
LIN {X 0,Y 43.457,Z 359.879,A -85,B 0,C 180,E1 -30271.888,E2 -30271.888} C_VEL
LIN {X 0,Y 37.128,Z 366.509,A -85,B 0,C 180,E1 -30280.782,E2 -30280.782} C_VEL
LIN {X 0,Y 31.056,Z 372.985,A -85,B 0,C 180,E1 -30295.542,E2 -30295.542} C_VEL
LIN {X 0,Y 27.766,Z 378.095,A -85,B 0,C 180,E1 -30315.335,E2 -30315.335} C_VEL
LIN {X 0,Y 27.451,Z 380.809,A -85,B 0,C 180,E1 -30329.997,E2 -30329.997} C_VEL
LIN {X 0,Y 27.932,Z 382.985,A -85,B 0,C 180,E1 -30344.57,E2 -30344.57} C_VEL
LIN {X 0,Y 29.766,Z 384.711,A -85,B 0,C 180,E1 -30358.175,E2 -30358.175} C_VEL
LIN {X 0,Y 37.315,Z 386.906,A -85,B 0,C 180,E1 -30378.88,E2 -30378.88} C_VEL
LIN {X 0,Y 48.089,Z 387.63,A -85,B 0,C 180,E1 -30391.265,E2 -30391.265} C_VEL
LIN {X 0,Y 54.056,Z 387.427,A -85,B 0,C 180,E1 -30395.517,E2 -30395.517} C_VEL
LIN {X 0,Y 66.663,Z 385.848,A -85,B 0,C 180,E1 -30401.591,E2 -30401.591} C_VEL
LIN {X 0,Y 79.798,Z 382.755,A -85,B 0,C 180,E1 -30405.646,E2 -30405.646} C_VEL
LIN {X 0,Y 89.89,Z 379.306,A -85,B 0,C 180,E1 -30407.77,E2 -30407.77} C_VEL
LIN {X 0,Y 100.098,Z 374.82,A -85,B 0,C 180,E1 -30409.406,E2 -30409.406} C_VEL
LIN {X 0,Y 106.955,Z 371.185,A -85,B 0,C 180,E1 -30410.28,E2 -30410.28} C_VEL
LIN {X 0,Y 109.857,Z 369.449,A -85,B 0,C 180,E1 -30411.268,E2 -30411.268} C_VEL
LIN {X 0,Y 99.16,Z 375.083,A -85,B 0,C 180,E1 -30412.864,E2 -30412.864} C_VEL
LIN {X 0,Y 86.306,Z 380.26,A -85,B 0,C 180,E1 -30415.327,E2 -30415.327} C_VEL
LIN {X 0,Y 77.376,Z 382.885,A -85,B 0,C 180,E1 -30417.591,E2 -30417.591} C_VEL
LIN {X 0,Y 69.857,Z 384.566,A -85,B 0,C 180,E1 -30419.997,E2 -30419.997} C_VEL
LIN {X 0,Y 63.315,Z 385.572,A -85,B 0,C 180,E1 -30422.57,E2 -30422.57} C_VEL
LIN {X 0,Y 54.105,Z 386.354,A -85,B 0,C 180,E1 -30427.459,E2 -30427.459} C_VEL
LIN {X 0,Y 43.822,Z 386.153,A -85,B 0,C 180,E1 -30435.796,E2 -30435.796} C_VEL
LIN {X 0,Y 39.066,Z 385.586,A -85,B 0,C 180,E1 -30441.673,E2 -30441.673} C_VEL
LIN {X 0,Y 34.611,Z 384.812,A -85,B 0,C 180,E1 -30447.592,E2 -30447.592} C_VEL
LIN {X 0,Y 26.893,Z 382.944,A -85,B 0,C 180,E1 -30458.782,E2 -30458.782} C_VEL
LIN {X 0,Y 21.738,Z 380.903,A -85,B 0,C 180,E1 -30472.426,E2 -30472.426} C_VEL
LIN {X 0,Y 19.751,Z 379.009,A -85,B 0,C 180,E1 -30487.051,E2 -30487.051} C_VEL
LIN {X 0,Y 19.658,Z 378.309,A -85,B 0,C 180,E1 -30492.438,E2 -30492.438} C_VEL
LIN {X 0,Y 22.424,Z 373.834,A -85,B 0,C 180,E1 -30520.205,E2 -30520.205} C_VEL
LIN {X 0,Y 28.577,Z 368.115,A -85,B 0,C 180,E1 -30539.466,E2 -30539.466} C_VEL
LIN {X 0,Y 35.428,Z 362.033,A -85,B 0,C 180,E1 -30550.151,E2 -30550.151} C_VEL
LIN {X 0,Y 42.93,Z 354.748,A -85,B 0,C 180,E1 -30557.453,E2 -30557.453} C_VEL
LIN {X 0,Y 50.894,Z 345.889,A -85,B 0,C 180,E1 -30562.565,E2 -30562.565} C_VEL
LIN {X 0,Y 59.133,Z 334.946,A -85,B 0,C 180,E1 -30566.303,E2 -30566.303} C_VEL
LIN {X 0,Y 65.788,Z 324.063,A -85,B 0,C 180,E1 -30568.721,E2 -30568.721} C_VEL
LIN {X 0,Y 71.704,Z 311.764,A -85,B 0,C 180,E1 -30570.498,E2 -30570.498} C_VEL
LIN {X 0,Y 76.326,Z 299.073,A -85,B 0,C 180,E1 -30571.714,E2 -30571.714} C_VEL
LIN {X 0,Y 79.543,Z 286.234,A -85,B 0,C 180,E1 -30572.57,E2 -30572.57} C_VEL
LIN {X 0,Y 82.081,Z 268.873,A -85,B 0,C 180,E1 -30573.12,E2 -30573.12} C_VEL
LIN {X 0,Y 82.739,Z 263.14,A -85,B 0,C 180,E1 -30573.375,E2 -30573.375} C_VEL
LIN {X 0,Y 81.558,Z 258.726,A -85,B 0,C 180,E1 -30578.487,E2 -30578.487} C_VEL
LIN {X 0,Y 80.83,Z 255.8,A -85,B 0,C 180,E1 -30583.862,E2 -30583.862} C_VEL
LIN {X 0,Y 80.561,Z 254.827,A -85,B 0,C 180,E1 -30589.955,E2 -30589.955} C_VEL
LIN {X 0,Y 80.881,Z 255.074,A -85,B 0,C 180,E1 -30595.339,E2 -30595.339} C_VEL
LIN {X 0,Y 81.449,Z 257.986,A -85,B 0,C 180,E1 -30600.216,E2 -30600.216} C_VEL
LIN {X 0,Y 82.476,Z 261.962,A -85,B 0,C 180,E1 -30605.044,E2 -30605.044} C_VEL
LIN {X 0,Y 82.802,Z 263.399,A -85,B 0,C 180,E1 -30606.322,E2 -30606.322} C_VEL
LIN {X 0,Y 79.927,Z 285.329,A -85,B 0,C 180,E1 -30607.073,E2 -30607.073} C_VEL
LIN {X 0,Y 76.679,Z 298.979,A -85,B 0,C 180,E1 -30607.733,E2 -30607.733} C_VEL
LIN {X 0,Y 72.425,Z 311.143,A -85,B 0,C 180,E1 -30608.66,E2 -30608.66} C_VEL
LIN {X 0,Y 66.922,Z 322.969,A -85,B 0,C 180,E1 -30610.077,E2 -30610.077} C_VEL
LIN {X 0,Y 60.211,Z 334.372,A -85,B 0,C 180,E1 -30612.154,E2 -30612.154} C_VEL
LIN {X 0,Y 53.591,Z 343.586,A -85,B 0,C 180,E1 -30614.732,E2 -30614.732} C_VEL
LIN {X 0,Y 46.153,Z 352.363,A -85,B 0,C 180,E1 -30618.636,E2 -30618.636} C_VEL
LIN {X 0,Y 37.177,Z 361.473,A -85,B 0,C 180,E1 -30626.104,E2 -30626.104} C_VEL
LIN {X 0,Y 28.938,Z 368.907,A -85,B 0,C 180,E1 -30637.874,E2 -30637.874} C_VEL
LIN {X 0,Y 23.588,Z 373.937,A -85,B 0,C 180,E1 -30653.419,E2 -30653.419} C_VEL
LIN {X 0,Y 20.382,Z 378.774,A -85,B 0,C 180,E1 -30680.069,E2 -30680.069} C_VEL
LIN {X 0,Y 20.349,Z 380.125,A -85,B 0,C 180,E1 -30689.996,E2 -30689.996} C_VEL
LIN {X 0,Y 21.136,Z 382.361,A -85,B 0,C 180,E1 -30709.418,E2 -30709.418} C_VEL
LIN {X 0,Y 23.746,Z 384.153,A -85,B 0,C 180,E1 -30726.291,E2 -30726.291} C_VEL
LIN {X 0,Y 27.898,Z 385.54,A -85,B 0,C 180,E1 -30739.087,E2 -30739.087} C_VEL
LIN {X 0,Y 38.907,Z 387.109,A -85,B 0,C 180,E1 -30754.576,E2 -30754.576} C_VEL
LIN {X 0,Y 51.517,Z 387.21,A -85,B 0,C 180,E1 -30762.733,E2 -30762.733} C_VEL
LIN {X 0,Y 63.549,Z 385.99,A -85,B 0,C 180,E1 -30767.218,E2 -30767.218} C_VEL
LIN {X 0,Y 71.531,Z 384.485,A -85,B 0,C 180,E1 -30769.266,E2 -30769.266} C_VEL
LIN {X 0,Y 78.341,Z 382.803,A -85,B 0,C 180,E1 -30770.681,E2 -30770.681} C_VEL
LIN {X 0,Y 78.079,Z 382.815,A -85,B 0,C 180,E1 -30771.936,E2 -30771.936} C_VEL
LIN {X 0,Y 68.636,Z 384.888,A -85,B 0,C 180,E1 -30774.12,E2 -30774.12} C_VEL
LIN {X 0,Y 56.253,Z 386.398,A -85,B 0,C 180,E1 -30778.128,E2 -30778.128} C_VEL
LIN {X 0,Y 49.21,Z 386.673,A -85,B 0,C 180,E1 -30781.418,E2 -30781.418} C_VEL
LIN {X 0,Y 42.378,Z 386.52,A -85,B 0,C 180,E1 -30785.714,E2 -30785.714} C_VEL
LIN {X 0,Y 34.502,Z 385.636,A -85,B 0,C 180,E1 -30793.148,E2 -30793.148} C_VEL
LIN {X 0,Y 24.744,Z 383.282,A -85,B 0,C 180,E1 -30811.567,E2 -30811.567} C_VEL
LIN {X 0,Y 20.075,Z 380.088,A -85,B 0,C 180,E1 -30838.327,E2 -30838.327} C_VEL
LIN {X 0,Y 19.658,Z 378.309,A -85,B 0,C 180,E1 -30852.438,E2 -30852.438} C_VEL
LIN {X 0,Y 19.9,Z 376.129,A -85,B 0,C 180,E1 -30868.281,E2 -30868.281} C_VEL
LIN {X 0,Y 20.562,Z 373.69,A -85,B 0,C 180,E1 -30883.575,E2 -30883.575} C_VEL
LIN {X 0,Y 25.699,Z 367.08,A -85,B 0,C 180,E1 -30911.84,E2 -30911.84} C_VEL
LIN {X 0,Y 29.562,Z 363.753,A -85,B 0,C 180,E1 -30918.365,E2 -30918.365} C_VEL
LIN {X 0,Y 38.565,Z 355.953,A -85,B 0,C 180,E1 -30925.596,E2 -30925.596} C_VEL
LIN {X 0,Y 46.85,Z 347.541,A -85,B 0,C 180,E1 -30929.61,E2 -30929.61} C_VEL
LIN {X 0,Y 54.583,Z 338.138,A -85,B 0,C 180,E1 -30932.281,E2 -30932.281} C_VEL
LIN {X 0,Y 62.347,Z 326.429,A -85,B 0,C 180,E1 -30934.397,E2 -30934.397} C_VEL
LIN {X 0,Y 68.443,Z 314.882,A -85,B 0,C 180,E1 -30935.712,E2 -30935.712} C_VEL
LIN {X 0,Y 72.793,Z 304.233,A -85,B 0,C 180,E1 -30936.63,E2 -30936.63} C_VEL
LIN {X 0,Y 76.671,Z 291.273,A -85,B 0,C 180,E1 -30937.353,E2 -30937.353} C_VEL
LIN {X 0,Y 79.275,Z 277.565,A -85,B 0,C 180,E1 -30937.788,E2 -30937.788} C_VEL
LIN {X 0,Y 80.596,Z 266.966,A -85,B 0,C 180,E1 -30938.084,E2 -30938.084} C_VEL
LIN {X 0,Y 80.022,Z 264.043,A -85,B 0,C 180,E1 -30942.245,E2 -30942.245} C_VEL
LIN {X 0,Y 79.751,Z 262.504,A -85,B 0,C 180,E1 -30945.787,E2 -30945.787} C_VEL
LIN {X 0,Y 79.686,Z 261.91,A -85,B 0,C 180,E1 -30951.62,E2 -30951.62} C_VEL
LIN {X 0,Y 79.87,Z 262.192,A -85,B 0,C 180,E1 -30954.553,E2 -30954.553} C_VEL
LIN {X 0,Y 80.283,Z 265.147,A -85,B 0,C 180,E1 -30959.242,E2 -30959.242} C_VEL
LIN {X 0,Y 80.653,Z 266.994,A -85,B 0,C 180,E1 -30961.605,E2 -30961.605} C_VEL
LIN {X 0,Y 77.829,Z 286.853,A -85,B 0,C 180,E1 -30962.146,E2 -30962.146} C_VEL
LIN {X 0,Y 74.522,Z 299.864,A -85,B 0,C 180,E1 -30962.61,E2 -30962.61} C_VEL
LIN {X 0,Y 69.524,Z 313.17,A -85,B 0,C 180,E1 -30963.373,E2 -30963.373} C_VEL
LIN {X 0,Y 63.446,Z 325.32,A -85,B 0,C 180,E1 -30964.457,E2 -30964.457} C_VEL
LIN {X 0,Y 56.533,Z 336.14,A -85,B 0,C 180,E1 -30965.979,E2 -30965.979} C_VEL
LIN {X 0,Y 49.064,Z 345.737,A -85,B 0,C 180,E1 -30968.24,E2 -30968.24} C_VEL
LIN {X 0,Y 41.219,Z 354.12,A -85,B 0,C 180,E1 -30971.349,E2 -30971.349} C_VEL
LIN {X 0,Y 31.416,Z 363.029,A -85,B 0,C 180,E1 -30978.048,E2 -30978.048} C_VEL
LIN {X 0,Y 22.291,Z 370.077,A -85,B 0,C 180,E1 -30989.879,E2 -30989.879} C_VEL
LIN {X 0,Y 14.456,Z 376.51,A -85,B 0,C 180,E1 -31020.906,E2 -31020.906} C_VEL
LIN {X 0,Y 13.266,Z 379.439,A -85,B 0,C 180,E1 -31049.995,E2 -31049.995} C_VEL
LIN {X 0,Y 14.633,Z 381.738,A -85,B 0,C 180,E1 -31078.699,E2 -31078.699} C_VEL
LIN {X 0,Y 18.51,Z 383.588,A -85,B 0,C 180,E1 -31099.402,E2 -31099.402} C_VEL
LIN {X 0,Y 29.937,Z 386.105,A -85,B 0,C 180,E1 -31119.884,E2 -31119.884} C_VEL
LIN {X 0,Y 43.088,Z 387.054,A -85,B 0,C 180,E1 -31128.134,E2 -31128.134} C_VEL
LIN {X 0,Y 49.871,Z 386.978,A -85,B 0,C 180,E1 -31130.556,E2 -31130.556} C_VEL
LIN {X 0,Y 50.927,Z 386.904,A -85,B 0,C 180,E1 -31132.063,E2 -31132.063} C_VEL
LIN {X 0,Y 42.312,Z 386.837,A -85,B 0,C 180,E1 -31135.262,E2 -31135.262} C_VEL
LIN {X 0,Y 34.063,Z 386.168,A -85,B 0,C 180,E1 -31139.994,E2 -31139.994} C_VEL
LIN {X 0,Y 21.737,Z 383.849,A -85,B 0,C 180,E1 -31154.095,E2 -31154.095} C_VEL
LIN {X 0,Y 14.184,Z 380.786,A -85,B 0,C 180,E1 -31182,E2 -31182} C_VEL
LIN {X 0,Y 13.307,Z 376.613,A -85,B 0,C 180,E1 -31230.005,E2 -31230.005} C_VEL
LIN {X 0,Y 19.695,Z 371.239,A -85,B 0,C 180,E1 -31262.366,E2 -31262.366} C_VEL
LIN {X 0,Y 29.562,Z 363.753,A -85,B 0,C 180,E1 -31278.365,E2 -31278.365} C_VEL
LIN {X 0,Y 33.494,Z 360.266,A -85,B 0,C 180,E1 -31283.342,E2 -31283.342} C_VEL
LIN {X 0,Y 39.364,Z 354.188,A -85,B 0,C 180,E1 -31291.65,E2 -31291.65} C_VEL
LIN {X 0,Y 45.322,Z 347.529,A -85,B 0,C 180,E1 -31297.535,E2 -31297.535} C_VEL
LIN {X 0,Y 49.067,Z 343.124,A -85,B 0,C 180,E1 -31299.028,E2 -31299.028} C_VEL
LIN {X 0,Y 56.92,Z 332.809,A -85,B 0,C 180,E1 -31300.304,E2 -31300.304} C_VEL
LIN {X 0,Y 64.109,Z 321.004,A -85,B 0,C 180,E1 -31301.256,E2 -31301.256} C_VEL
LIN {X 0,Y 69.723,Z 309.124,A -85,B 0,C 180,E1 -31302.002,E2 -31302.002} C_VEL
LIN {X 0,Y 74.301,Z 295.891,A -85,B 0,C 180,E1 -31302.475,E2 -31302.475} C_VEL
LIN {X 0,Y 77.332,Z 282.853,A -85,B 0,C 180,E1 -31302.846,E2 -31302.846} C_VEL
LIN {X 0,Y 78.97,Z 271.133,A -85,B 0,C 180,E1 -31303.086,E2 -31303.086} C_VEL
LIN {X 0,Y 78.806,Z 269.468,A -85,B 0,C 180,E1 -31306.439,E2 -31306.439} C_VEL
LIN {X 0,Y 78.781,Z 268.951,A -85,B 0,C 180,E1 -31311.523,E2 -31311.523} C_VEL
LIN {X 0,Y 78.873,Z 269.279,A -85,B 0,C 180,E1 -31313.669,E2 -31313.669} C_VEL
LIN {X 0,Y 78.998,Z 271.097,A -85,B 0,C 180,E1 -31316.575,E2 -31316.575} C_VEL
LIN {X 0,Y 76.539,Z 287.336,A -85,B 0,C 180,E1 -31316.966,E2 -31316.966} C_VEL
LIN {X 0,Y 73.193,Z 300.033,A -85,B 0,C 180,E1 -31317.206,E2 -31317.206} C_VEL
LIN {X 0,Y 68.146,Z 313.185,A -85,B 0,C 180,E1 -31317.581,E2 -31317.581} C_VEL
LIN {X 0,Y 62.411,Z 324.485,A -85,B 0,C 180,E1 -31318.066,E2 -31318.066} C_VEL
LIN {X 0,Y 55.359,Z 335.454,A -85,B 0,C 180,E1 -31318.833,E2 -31318.833} C_VEL
LIN {X 0,Y 47.489,Z 345.328,A -85,B 0,C 180,E1 -31320.005,E2 -31320.005} C_VEL
LIN {X 0,Y 38.674,Z 354.388,A -85,B 0,C 180,E1 -31321.791,E2 -31321.791} C_VEL
LIN {X 0,Y 28.255,Z 363.184,A -85,B 0,C 180,E1 -31325.738,E2 -31325.738} C_VEL
LIN {X 0,Y 18.068,Z 370.144,A -85,B 0,C 180,E1 -31333.46,E2 -31333.46} C_VEL
LIN {X 0,Y 8.929,Z 375.695,A -85,B 0,C 180,E1 -31358.072,E2 -31358.072} C_VEL
LIN {X 0,Y 6.162,Z 378.703,A -85,B 0,C 180,E1 -31409.988,E2 -31409.988} C_VEL
LIN {X 0,Y 9.078,Z 381.115,A -85,B 0,C 180,E1 -31460.718,E2 -31460.718} C_VEL
LIN {X 0,Y 21.466,Z 384.529,A -85,B 0,C 180,E1 -31489.166,E2 -31489.166} C_VEL
LIN {X 0,Y 21.214,Z 384.409,A -85,B 0,C 180,E1 -31493.624,E2 -31493.624} C_VEL
LIN {X 0,Y 10.71,Z 381.475,A -85,B 0,C 180,E1 -31510.193,E2 -31510.193} C_VEL
LIN {X 0,Y 5.811,Z 377.43,A -85,B 0,C 180,E1 -31590.012,E2 -31590.012} C_VEL
LIN {X 0,Y 14.013,Z 372.2,A -85,B 0,C 180,E1 -31638.799,E2 -31638.799} C_VEL
LIN {X 0,Y 24.281,Z 365.666,A -85,B 0,C 180,E1 -31650.271,E2 -31650.271} C_VEL
LIN {X 0,Y 33.731,Z 358.409,A -85,B 0,C 180,E1 -31654.947,E2 -31654.947} C_VEL
LIN {X 0,Y 43.625,Z 349.124,A -85,B 0,C 180,E1 -31657.876,E2 -31657.876} C_VEL
LIN {X 0,Y 49.067,Z 343.124,A -85,B 0,C 180,E1 -31659.028,E2 -31659.028} C_VEL
LIN {X 0,Y 52.653,Z 338.595,A -85,B 0,C 180,E1 -31660.272,E2 -31660.272} C_VEL
LIN {X 0,Y 57.847,Z 330.89,A -85,B 0,C 180,E1 -31663.796,E2 -31663.796} C_VEL
LIN {X 0,Y 62.646,Z 322.787,A -85,B 0,C 180,E1 -31666.864,E2 -31666.864} C_VEL
LIN {X 0,Y 65.376,Z 317.558,A -85,B 0,C 180,E1 -31667.617,E2 -31667.617} C_VEL
LIN {X 0,Y 70.423,Z 306.075,A -85,B 0,C 180,E1 -31667.852,E2 -31667.852} C_VEL
LIN {X 0,Y 74.661,Z 292.89,A -85,B 0,C 180,E1 -31667.957,E2 -31667.957} C_VEL
LIN {X 0,Y 77.3,Z 280.037,A -85,B 0,C 180,E1 -31668.115,E2 -31668.115} C_VEL
LIN {X 0,Y 77.842,Z 276.282,A -85,B 0,C 180,E1 -31668.285,E2 -31668.285} C_VEL
LIN {X 0,Y 77.88,Z 275.986,A -85,B 0,C 180,E1 -31671.513,E2 -31671.513} C_VEL
LIN {X 0,Y 75.712,Z 288.633,A -85,B 0,C 180,E1 -31671.661,E2 -31671.661} C_VEL
LIN {X 0,Y 72.177,Z 301.247,A -85,B 0,C 180,E1 -31671.643,E2 -31671.643} C_VEL
LIN {X 0,Y 67.49,Z 313.198,A -85,B 0,C 180,E1 -31671.608,E2 -31671.608} C_VEL
LIN {X 0,Y 61.287,Z 325.211,A -85,B 0,C 180,E1 -31671.526,E2 -31671.526} C_VEL
LIN {X 0,Y 53.309,Z 337.128,A -85,B 0,C 180,E1 -31671.417,E2 -31671.417} C_VEL
LIN {X 0,Y 45.474,Z 346.563,A -85,B 0,C 180,E1 -31671.413,E2 -31671.413} C_VEL
LIN {X 0,Y 37.337,Z 354.653,A -85,B 0,C 180,E1 -31671.212,E2 -31671.212} C_VEL
LIN {X 0,Y 28.443,Z 362.016,A -85,B 0,C 180,E1 -31671.268,E2 -31671.268} C_VEL
LIN {X 0,Y 17.817,Z 369.188,A -85,B 0,C 180,E1 -31670.475,E2 -31670.475} C_VEL
LIN {X 0,Y 14.275,Z 371.228,A -85,B 0,C 180,E1 -31669.985,E2 -31669.985} C_VEL
LIN {X 0,Y 14.353,Z 371.172,A -85,B 0,C 180,E1 -31668.342,E2 -31668.342} C_VEL
LIN {X 0,Y 25.244,Z 364.286,A -85,B 0,C 180,E1 -31667.02,E2 -31667.02} C_VEL
LIN {X 0,Y 36.049,Z 355.773,A -85,B 0,C 180,E1 -31667.117,E2 -31667.117} C_VEL
LIN {X 0,Y 46.104,Z 345.798,A -85,B 0,C 180,E1 -31667.234,E2 -31667.234} C_VEL
